(* IEC 61131-3 sources: SmartHomeNew/snapshots/2026-05-25 (part 3) *)

(* ---- FB_Heating_RootCause_Diagnostics.st ---- *)
// ==============================================================================
// Heating root-cause diagnostics observer
// Public diagnostics/explainability layer.
// Does NOT own control/runtime decisions.
// ==============================================================================
FUNCTION_BLOCK FB_Heating_RootCause_Diagnostics
VAR_INPUT
    VI_Enable : BOOL;
END_VAR
VAR
    fbRootCause : FB_Diagnostics_RootCause;
    fbDemandMap : FB_Heating_Demand_Map;
    L_Demand_Map : ARRAY[1..GVL_CONSTANTS.C_MAX_MANIFOLDS] OF BOOL;
END_VAR

IF NOT VI_Enable THEN
    GVL_STATE.G_Heating_RootCause := E_Heating_RootCause.RC_NONE;
    GVL_STATE.G_Heating_RootConfidence := 0.0;
    GVL_STATE.G_Heating_Confidence := 0.0;
    GVL_STATE.G_Heating_Error_Score := 1.0;
    GVL_STATE.G_Heating_Confidence_Reason_Code := -1;
    GVL_STATE.G_Heating_Confidence_Reason_Text := 'Heating diagnostics disabled';
    RETURN;
END_IF;

// ======================================================
// DEMAND MAP
// ======================================================
fbDemandMap(
    VI_Zone_Valves := GVL_STATE.G_Zone_Valves,
    VI_Zone_Configs := GVL_CONFIG.G_HMI_FloorHeating_Configs,
    VO_Manifold_Demand_Map => L_Demand_Map
);

// ======================================================
// INTERNAL INFERENCE ENGINE
// ======================================================
fbRootCause(
    VI_Emergency_Stop := GVL_STATE.G_Safety_Emergency_Stop,
    VI_Gas_Safety := GVL_STATE.G_Safety_Gas_Latched,
    VI_IO_Failsafe := GVL_STATE.G_Heating_IO_Fault,

    VI_Cascade_Available := GVL_STATE.G_Heating_Cascade_Available,
    VI_Cascade_Degraded := GVL_STATE.G_Heating_Cascade_Degraded,
    VI_Cascade_Partial_Capacity := GVL_STATE.G_Heating_Cascade_Partial_Capacity,
    VI_Cascade_No_Flame := GVL_STATE.G_Heating_Cascade_No_Flame,
    VI_Cascade_Transport_Degraded := GVL_STATE.G_Heating_Cascade_Transport_Degraded,
    VI_Cascade_Ignition_Timeout := GVL_STATE.G_Heating_Cascade_Ignition_Timeout,
    VI_Cascade_Active_Boilers := GVL_STATE.G_Heating_Cascade_Active_Boilers,
    VI_Cascade_Available_Boilers := GVL_STATE.G_Heating_Cascade_Available_Boilers,

    VI_Boiler_OT_Online := GVL_STATE.G_Boiler_OT_Online,
    VI_Boiler_Error := GVL_STATE.G_Boiler_Error,
    VI_Boiler_Flame := GVL_STATE.G_Boiler_Flame,
    VI_Boiler_OT_Command_Timeout := GVL_STATE.G_Boiler_OT_Command_Timeout,
    VI_Boiler_OT_Heartbeat_Timeout := GVL_STATE.G_Boiler_OT_Heartbeat_Timeout,
    VI_Boiler_OT_Adapter_Error := GVL_STATE.G_Boiler_OT_Adapter_Error,

    VI_Manifold_Pumps := GVL_STATE.G_Manifold_Pumps,
    VI_Manifold_Valves := GVL_STATE.G_Manifold_Valves,

    VI_Sensor_Error := GVL_STATE.G_Heating_Sensor_Fault,
    VI_Supply_Temps := GVL_STATE.G_Manifold_T_Supply,
    VI_Target_Supply := GVL_STATE.G_Target_Temperature,
    VI_Demand_Map := L_Demand_Map
);

// ======================================================
// PUBLIC DIAGNOSTICS STATE
// ======================================================
GVL_STATE.G_Heating_RootCause := fbRootCause.VO_RootCause;
GVL_STATE.G_Heating_RootConfidence := fbRootCause.VO_Confidence;
GVL_STATE.G_Heating_Confidence := fbRootCause.VO_Confidence;
GVL_STATE.G_Heating_Error_Score := fbRootCause.VO_Error_Score;
GVL_STATE.G_Heating_Confidence_Reason_Code := fbRootCause.VO_Reason_Code;
GVL_STATE.G_Heating_Confidence_Reason_Text := fbRootCause.VO_Reason_Text;

END_FUNCTION_BLOCK
// >>> BULK_SYNC_ANCHOR: FB_Heating_RootCause_Diagnostics <<<

(* ---- FB_Heating_Runtime_Event_Manager.st ---- *)
// ==============================================================================
// Heating runtime event manager
// Read-only orchestration telemetry/event layer.
// DOES NOT own runtime.
// DOES NOT own heating logic.
// DOES NOT own diagnostics.
// DOES NOT own OpenTherm transport.
// ==============================================================================
FUNCTION_BLOCK FB_Heating_Runtime_Event_Manager
VAR_INPUT
    VI_Enable : BOOL;
    VI_Event : ST_Heating_Runtime_Phase_Event;
END_VAR
VAR_IN_OUT
    VIO_Buffer : ST_Heating_Runtime_Event_Buffer;
END_VAR
VAR_OUTPUT
    VO_Event_Stored : BOOL;
    VO_Buffer_Overflow : BOOL;
    VO_Manager_Ready : BOOL;
    VO_Manager_Status_Code : UINT;
    VO_Manager_Status_Text : STRING(128);
END_VAR
VAR
    L_Write_Index : UINT;
END_VAR

// ======================================================
// DEFAULTS
// ======================================================
VO_Event_Stored := FALSE;
VO_Buffer_Overflow := FALSE;
VO_Manager_Ready := FALSE;
VO_Manager_Status_Code := 0;
VO_Manager_Status_Text := 'Heating runtime event manager disabled';

IF NOT VI_Enable THEN
    RETURN;
END_IF;

// ======================================================
// BUFFER VALIDATION
// ======================================================
IF VIO_Buffer.Write_Index > 32 THEN
    VIO_Buffer.Write_Index := 1;
END_IF;

IF VIO_Buffer.Read_Index > 32 THEN
    VIO_Buffer.Read_Index := 1;
END_IF;

// ======================================================
// WRITE INDEX
// ======================================================
L_Write_Index := VIO_Buffer.Write_Index + 1;

IF L_Write_Index > 32 THEN
    L_Write_Index := 1;
END_IF;

// ======================================================
// STORE EVENT
// ======================================================
VIO_Buffer.Events[L_Write_Index] := VI_Event;
VIO_Buffer.Write_Index := L_Write_Index;

IF VIO_Buffer.Event_Count < 32 THEN
    VIO_Buffer.Event_Count := VIO_Buffer.Event_Count + 1;
ELSE
    VIO_Buffer.Overflow := TRUE;
    VO_Buffer_Overflow := TRUE;
END_IF;

// ======================================================
// BUFFER INTEGRITY
// ======================================================
VIO_Buffer.Ordering_Integrity_Valid :=
    VI_Event.Ordering_Valid;

VIO_Buffer.Isolation_Integrity_Valid :=
    VI_Event.Isolation_Valid;

VIO_Buffer.Diagnostics_Visibility_Valid :=
    VI_Event.Diagnostics_Visible;

VIO_Buffer.Explainability_Visibility_Valid :=
    VI_Event.Explainability_Visible;

VIO_Buffer.OpenTherm_Ownership_Valid :=
    VI_Event.OpenTherm_Ownership_Valid;

VIO_Buffer.Cascade_Ownership_Valid :=
    VI_Event.Cascade_Ownership_Valid;

VIO_Buffer.Safety_Ownership_Valid :=
    VI_Event.Safety_Integrity_Valid;

VIO_Buffer.Lifecycle_Integrity_Valid :=
    NOT VI_Event.Event_Failed;

// ======================================================
// BUFFER STATUS
// ======================================================
IF VO_Buffer_Overflow THEN
    VIO_Buffer.Status_Code := 100;
    VIO_Buffer.Status_Text := 'Heating runtime event buffer overflow';
ELSE
    VIO_Buffer.Status_Code := 1;
    VIO_Buffer.Status_Text := 'Heating runtime event stored';
END_IF;

// ======================================================
// OUTPUT STATUS
// ======================================================
VO_Event_Stored := TRUE;
VO_Manager_Ready := TRUE;
VO_Manager_Status_Code := VIO_Buffer.Status_Code;
VO_Manager_Status_Text := VIO_Buffer.Status_Text;

END_FUNCTION_BLOCK
// >>> BULK_SYNC_ANCHOR: FB_Heating_Runtime_Event_Manager <<<

(* ---- FB_Heating_Runtime_Observer.st ---- *)
// ==============================================================================
// Heating runtime observer
// Minimal observer-only runtime attachment.
// Read-only.
// Governance-locked.
// Finalized-state observation only.
// ==============================================================================
FUNCTION_BLOCK FB_Heating_Runtime_Observer
VAR_INPUT
    VI_Enable : BOOL;
    VI_Runtime_Context : ST_Heating_Runtime_Context;
    VI_Diagnostics_Valid : BOOL;
END_VAR
VAR_OUTPUT
    VO_Observation : ST_Heating_Runtime_Observation;

    VO_Observer_Ready : BOOL;
    VO_Observer_Fault : BOOL;
    VO_Status_Code : UINT;
    VO_Status_Text : STRING(128);
END_VAR

// ======================================================
// DEFAULTS
// ======================================================
VO_Observation.Runtime_Active := FALSE;
VO_Observation.Runtime_Ready := FALSE;
VO_Observation.Runtime_Fault := FALSE;
VO_Observation.Current_Phase := E_Heating_Runtime_Phase.HRP_DISABLED;

VO_Observation.DHW_Demand_Active := FALSE;
VO_Observation.DHW_Heating_Active := FALSE;
VO_Observation.DHW_Circulation_Active := FALSE;

VO_Observation.Heating_Demand_Active := FALSE;
VO_Observation.Heating_Runtime_Active := FALSE;
VO_Observation.Heating_Output_Active := FALSE;

VO_Observation.Cascade_Available := FALSE;
VO_Observation.Cascade_Degraded := FALSE;
VO_Observation.Cascade_Active_Boilers := 0;
VO_Observation.Cascade_Available_Boilers := 0;

VO_Observation.OpenTherm_Online := FALSE;
VO_Observation.OpenTherm_Command_Valid := FALSE;
VO_Observation.OpenTherm_Transport_Degraded := FALSE;

VO_Observation.Diagnostics_Active := FALSE;
VO_Observation.Explainability_Active := FALSE;

VO_Observation.DHW_Before_Heating_Observed := FALSE;
VO_Observation.Diagnostics_After_Publication_Observed := FALSE;
VO_Observation.Output_Projection_Last_Observed := FALSE;

VO_Observation.Runtime_Ownership_Valid := TRUE;
VO_Observation.Diagnostics_Ownership_Valid := TRUE;
VO_Observation.OpenTherm_Ownership_Valid := TRUE;
VO_Observation.Cascade_Ownership_Valid := TRUE;
VO_Observation.Safety_Ownership_Valid := TRUE;

VO_Observation.Observation_Status_Code := 0;
VO_Observation.Observation_Status_Text := 'Heating runtime observer disabled';

VO_Observer_Ready := FALSE;
VO_Observer_Fault := FALSE;
VO_Status_Code := 0;
VO_Status_Text := 'Heating runtime observer disabled';

IF NOT VI_Enable THEN
    RETURN;
END_IF;

// ======================================================
// FINALIZED-STATE OBSERVATION ONLY
// ======================================================
VO_Observation.Runtime_Active := VI_Runtime_Context.Runtime_Enabled;
VO_Observation.Runtime_Ready := VI_Runtime_Context.Runtime_Ready;
VO_Observation.Runtime_Fault := VI_Runtime_Context.Runtime_Fault;
VO_Observation.Current_Phase := VI_Runtime_Context.Current_Phase;

VO_Observation.Diagnostics_Active := VI_Diagnostics_Valid;
VO_Observation.Explainability_Active := VI_Runtime_Context.Explainability_Isolation_Valid;

VO_Observation.DHW_Before_Heating_Observed :=
    VI_Runtime_Context.DHW_Before_Heating_Valid;

VO_Observation.Diagnostics_After_Publication_Observed :=
    VI_Runtime_Context.State_Publication_Before_Diagnostics_Valid;

VO_Observation.Output_Projection_Last_Observed :=
    VI_Runtime_Context.Output_Projection_Last_Valid;

VO_Observation.Runtime_Ownership_Valid := TRUE;
VO_Observation.Diagnostics_Ownership_Valid :=
    VI_Runtime_Context.Diagnostics_Isolation_Valid;

VO_Observation.OpenTherm_Ownership_Valid :=
    VI_Runtime_Context.OpenTherm_Ownership_Valid;

VO_Observation.Cascade_Ownership_Valid :=
    VI_Runtime_Context.Cascade_Ownership_Valid;

VO_Observation.Safety_Ownership_Valid :=
    VI_Runtime_Context.Safety_Isolation_Valid;

// These domain-specific runtime values remain intentionally FALSE/0 here.
// They must be populated only by finalized publication contracts, not by internal runtime scans.
VO_Observation.DHW_Demand_Active := FALSE;
VO_Observation.DHW_Heating_Active := FALSE;
VO_Observation.DHW_Circulation_Active := FALSE;
VO_Observation.Heating_Demand_Active := FALSE;
VO_Observation.Heating_Runtime_Active := FALSE;
VO_Observation.Heating_Output_Active := FALSE;
VO_Observation.Cascade_Available := FALSE;
VO_Observation.Cascade_Degraded := FALSE;
VO_Observation.Cascade_Active_Boilers := 0;
VO_Observation.Cascade_Available_Boilers := 0;
VO_Observation.OpenTherm_Online := FALSE;
VO_Observation.OpenTherm_Command_Valid := FALSE;
VO_Observation.OpenTherm_Transport_Degraded := FALSE;

// ======================================================
// STATUS
// ======================================================
IF VI_Runtime_Context.Runtime_Fault THEN
    VO_Observation.Observation_Status_Code := 900;
    VO_Observation.Observation_Status_Text := 'Heating runtime observer detected runtime fault';

ELSIF NOT VI_Diagnostics_Valid THEN
    VO_Observation.Observation_Status_Code := 200;
    VO_Observation.Observation_Status_Text := 'Heating runtime diagnostics publication invalid';

ELSE
    VO_Observation.Observation_Status_Code := 1;
    VO_Observation.Observation_Status_Text := 'Heating runtime observer nominal';
END_IF;

VO_Observer_Ready := TRUE;
VO_Observer_Fault := FALSE;

VO_Status_Code := VO_Observation.Observation_Status_Code;
VO_Status_Text := VO_Observation.Observation_Status_Text;

END_FUNCTION_BLOCK
// >>> BULK_SYNC_ANCHOR: FB_Heating_Runtime_Observer <<<

(* ---- FB_Heating_Runtime_Observer_Authorization.st ---- *)
// ==============================================================================
// Heating runtime observer authorization
// Governed passive-bootstrap authorization only.
// Read-only.
// Deterministic.
// ==============================================================================
FUNCTION_BLOCK FB_Heating_Runtime_Observer_Authorization
VAR_INPUT
    VI_Enable_Request : BOOL;

    VI_Bootstrap_Mode : BOOL;
    VI_Passive_Mode : BOOL;
    VI_ReadOnly_Mode : BOOL;

    VI_Governance_Locked : BOOL;
    VI_Runtime_Authority_Disabled : BOOL;
    VI_Writable_Exports_Disabled : BOOL;
END_VAR
VAR_OUTPUT
    VO_Enable_Authorized : BOOL;
    VO_Enable_Effective : BOOL;

    VO_Authorization_Valid : BOOL;

    VO_Status_Code : UINT;
    VO_Status_Text : STRING(128);
END_VAR

// ======================================================
// DEFAULTS
// ======================================================
VO_Enable_Authorized := FALSE;
VO_Enable_Effective := FALSE;
VO_Authorization_Valid := FALSE;

VO_Status_Code := 0;
VO_Status_Text := 'Heating runtime observer authorization inactive';

// ======================================================
// REQUEST VALIDATION
// ======================================================
IF NOT VI_Enable_Request THEN
    RETURN;
END_IF;

// ======================================================
// GOVERNANCE VALIDATION
// ======================================================
IF NOT VI_Bootstrap_Mode THEN
    VO_Status_Code := 100;
    VO_Status_Text := 'Bootstrap mode required for observer authorization';
    RETURN;
END_IF;

IF NOT VI_Passive_Mode THEN
    VO_Status_Code := 110;
    VO_Status_Text := 'Passive mode required for observer authorization';
    RETURN;
END_IF;

IF NOT VI_ReadOnly_Mode THEN
    VO_Status_Code := 120;
    VO_Status_Text := 'Read-only mode required for observer authorization';
    RETURN;
END_IF;

IF NOT VI_Governance_Locked THEN
    VO_Status_Code := 130;
    VO_Status_Text := 'Governance lock required for observer authorization';
    RETURN;
END_IF;

IF NOT VI_Runtime_Authority_Disabled THEN
    VO_Status_Code := 140;
    VO_Status_Text := 'Runtime authority isolation required';
    RETURN;
END_IF;

IF NOT VI_Writable_Exports_Disabled THEN
    VO_Status_Code := 150;
    VO_Status_Text := 'Writable exports must remain disabled';
    RETURN;
END_IF;

// ======================================================
// AUTHORIZED PASSIVE BOOTSTRAP ACTIVATION
// ======================================================
VO_Enable_Authorized := TRUE;
VO_Enable_Effective := TRUE;
VO_Authorization_Valid := TRUE;

VO_Status_Code := 1;
VO_Status_Text := 'Heating runtime observer authorization granted';

END_FUNCTION_BLOCK
// >>> BULK_SYNC_ANCHOR: FB_Heating_Runtime_Observer_Authorization <<<

(* ---- FB_Heating_Runtime_Observer_Phase.st ---- *)
// ==============================================================================
// Heating runtime observer phase
// Owns governed observer authorization and finalized-state observer publication.
// Does NOT own heating control or output decisions.
// ==============================================================================
FUNCTION_BLOCK FB_Heating_Runtime_Observer_Phase
VAR_INPUT
    VI_Authorization_Stage : BOOL;
    VI_Finalization_Stage : BOOL;
    VI_Runtime_Context : ST_Heating_Runtime_Context;
    VI_Diagnostics_Valid : BOOL;
END_VAR
VAR_OUTPUT
    VO_Authorization_Executed : BOOL;
    VO_Finalization_Executed : BOOL;
    VO_Observer_Valid : BOOL;
END_VAR
VAR
    fbRuntimeObserver : FB_Heating_Runtime_Observer;
    fbRuntimeObserverAuthorization : FB_Heating_Runtime_Observer_Authorization;
    L_Enable_Last : BOOL := FALSE;
    L_Activation_Stabilized : BOOL := FALSE;
END_VAR

VO_Authorization_Executed := FALSE;
VO_Finalization_Executed := FALSE;
VO_Observer_Valid := FALSE;

// ======================================================
// GOVERNED OBSERVER AUTHORIZATION EVALUATION
// ======================================================
IF VI_Authorization_Stage THEN

    GVL_Heating_Runtime_Observer.G_Runtime_Observer_Lifecycle_State :=
        E_Runtime_Observer_Lifecycle_State.ROS_AUTHORIZATION_PENDING;
    GVL_Heating_Runtime_Observation.G_Runtime_Observer_Lifecycle_State :=
        E_Runtime_Observer_Lifecycle_State.ROS_AUTHORIZATION_PENDING;
    GVL_Heating_Runtime_Observation.G_Runtime_Observer_Lifecycle_Code := 10;
    GVL_Heating_Runtime_Observation.G_Runtime_Observer_Lifecycle_Text :=
        'Heating runtime observer authorization pending';
    GVL_Heating_Runtime_Observation.G_Runtime_Observer_Commissioning_Active :=
        GVL_Heating_Runtime_Observer.G_Runtime_Observer_Enable_Request;

    fbRuntimeObserverAuthorization(
        VI_Enable_Request := GVL_Heating_Runtime_Observer.G_Runtime_Observer_Enable_Request,
        VI_Bootstrap_Mode := GVL_Heating_Runtime_Observer.G_Runtime_Observer_Bootstrap_Mode,
        VI_Passive_Mode := GVL_Heating_Runtime_Observer.G_Runtime_Observer_Passive_Mode,
        VI_ReadOnly_Mode := GVL_Heating_Runtime_Observer.G_Runtime_Observer_ReadOnly_Mode,
        VI_Governance_Locked := GVL_Heating_Runtime_Observer.G_Runtime_Observer_Governance_Locked,
        VI_Runtime_Authority_Disabled := GVL_Heating_Runtime_Observer.G_Runtime_Observer_Runtime_Authority_Disabled,
        VI_Writable_Exports_Disabled := GVL_Heating_Runtime_Observer.G_Runtime_Observer_Writable_Exports_Disabled
    );

    GVL_Heating_Runtime_Observer.G_Runtime_Observer_Enable_Authorized :=
        fbRuntimeObserverAuthorization.VO_Enable_Authorized;

    GVL_Heating_Runtime_Observer.G_Runtime_Observer_Enable_Effective :=
        fbRuntimeObserverAuthorization.VO_Enable_Effective;

    GVL_Heating_Runtime_Observer.G_Runtime_Observer_Authorization_Valid :=
        fbRuntimeObserverAuthorization.VO_Authorization_Valid;

    GVL_Heating_Runtime_Observer.G_Runtime_Observer_Authorization_Status_Code :=
        fbRuntimeObserverAuthorization.VO_Status_Code;

    GVL_Heating_Runtime_Observer.G_Runtime_Observer_Authorization_Status_Text :=
        fbRuntimeObserverAuthorization.VO_Status_Text;

    IF NOT GVL_Heating_Runtime_Observer.G_Runtime_Observer_Enable_Request THEN
        GVL_Heating_Runtime_Observer.G_Runtime_Observer_Lifecycle_State :=
            E_Runtime_Observer_Lifecycle_State.ROS_INACTIVE;
        GVL_Heating_Runtime_Observation.G_Runtime_Observer_Lifecycle_State :=
            E_Runtime_Observer_Lifecycle_State.ROS_INACTIVE;
        GVL_Heating_Runtime_Observation.G_Runtime_Observer_Lifecycle_Code := 0;
        GVL_Heating_Runtime_Observation.G_Runtime_Observer_Lifecycle_Text :=
            'Heating runtime observer inactive';
        GVL_Heating_Runtime_Observation.G_Runtime_Observer_Commissioning_Active := FALSE;
    ELSIF NOT GVL_Heating_Runtime_Observer.G_Runtime_Observer_Enable_Effective THEN
        GVL_Heating_Runtime_Observer.G_Runtime_Observer_Lifecycle_State :=
            E_Runtime_Observer_Lifecycle_State.ROS_AUTHORIZATION_DENIED;
        GVL_Heating_Runtime_Observation.G_Runtime_Observer_Lifecycle_State :=
            E_Runtime_Observer_Lifecycle_State.ROS_AUTHORIZATION_DENIED;
        GVL_Heating_Runtime_Observation.G_Runtime_Observer_Lifecycle_Code := 20;
        GVL_Heating_Runtime_Observation.G_Runtime_Observer_Lifecycle_Text :=
            'Heating runtime observer authorization denied';
    END_IF;

    VO_Authorization_Executed := TRUE;
END_IF;

// ======================================================
// GOVERNED FINALIZED-STATE RUNTIME OBSERVER
// ======================================================
IF VI_Finalization_Stage THEN

    IF GVL_Heating_Runtime_Observer.G_Runtime_Observer_Enable_Effective THEN

        GVL_Heating_Runtime_Observer.G_Runtime_Observer_Rollback_Validated := FALSE;

        IF NOT L_Enable_Last THEN
            L_Activation_Stabilized := FALSE;

            GVL_Heating_Runtime_Observer.G_Runtime_Observer_Lifecycle_State :=
                E_Runtime_Observer_Lifecycle_State.ROS_STABILIZATION;
            GVL_Heating_Runtime_Observation.G_Runtime_Observer_Lifecycle_State :=
                E_Runtime_Observer_Lifecycle_State.ROS_STABILIZATION;
            GVL_Heating_Runtime_Observation.G_Runtime_Observer_Lifecycle_Code := 30;
            GVL_Heating_Runtime_Observation.G_Runtime_Observer_Lifecycle_Text :=
                'Heating runtime observer stabilization active';

            GVL_Heating_Runtime_Observation.G_Runtime_Observer_Commissioning_Required := TRUE;
            GVL_Heating_Runtime_Observation.G_Runtime_Observer_Commissioning_Active := TRUE;
            GVL_Heating_Runtime_Observation.G_Runtime_Observer_Commissioning_Complete := FALSE;

            GVL_Heating_Runtime_Observation.G_Runtime_Observation_Publication_Valid := FALSE;
            GVL_Heating_Runtime_Observation.G_Runtime_Observation_Stabilization_Complete := FALSE;
            GVL_Heating_Runtime_Observation.G_Runtime_Observation_Operational := FALSE;

            GVL_Heating_Runtime_Observation.G_Runtime_Observation_Valid := FALSE;
            GVL_Heating_Runtime_Observation.G_Runtime_Observer_Ready := FALSE;
            GVL_Heating_Runtime_Observation.G_Runtime_Observer_Fault := FALSE;
            GVL_Heating_Runtime_Observation.G_Runtime_Observation_Status_Code := 100;
            GVL_Heating_Runtime_Observation.G_Runtime_Observation_Status_Text :=
                'Heating runtime observer stabilization cycle active';
        END_IF;

        fbRuntimeObserver(
            VI_Enable := TRUE,
            VI_Runtime_Context := VI_Runtime_Context,
            VI_Diagnostics_Valid := VI_Diagnostics_Valid
        );

        GVL_Heating_Runtime_Observation.G_Runtime_Observation :=
            fbRuntimeObserver.VO_Observation;

        IF L_Activation_Stabilized THEN
            GVL_Heating_Runtime_Observer.G_Runtime_Observer_Lifecycle_State :=
                E_Runtime_Observer_Lifecycle_State.ROS_OPERATIONAL;
            GVL_Heating_Runtime_Observation.G_Runtime_Observer_Lifecycle_State :=
                E_Runtime_Observer_Lifecycle_State.ROS_OPERATIONAL;
            GVL_Heating_Runtime_Observation.G_Runtime_Observer_Lifecycle_Code := 40;
            GVL_Heating_Runtime_Observation.G_Runtime_Observer_Lifecycle_Text :=
                'Heating runtime observer operational';

            GVL_Heating_Runtime_Observation.G_Runtime_Observer_Commissioning_Required := FALSE;
            GVL_Heating_Runtime_Observation.G_Runtime_Observer_Commissioning_Active := FALSE;
            GVL_Heating_Runtime_Observation.G_Runtime_Observer_Commissioning_Complete := TRUE;

            GVL_Heating_Runtime_Observation.G_Runtime_Observation_Publication_Valid := TRUE;
            GVL_Heating_Runtime_Observation.G_Runtime_Observation_Stabilization_Complete := TRUE;
            GVL_Heating_Runtime_Observation.G_Runtime_Observation_Operational := TRUE;

            GVL_Heating_Runtime_Observation.G_Runtime_Observation_Valid := TRUE;
            GVL_Heating_Runtime_Observation.G_Runtime_Observer_Ready :=
                fbRuntimeObserver.VO_Observer_Ready;
            GVL_Heating_Runtime_Observation.G_Runtime_Observer_Fault :=
                fbRuntimeObserver.VO_Observer_Fault;
            GVL_Heating_Runtime_Observation.G_Runtime_Observation_Status_Code :=
                fbRuntimeObserver.VO_Status_Code;
            GVL_Heating_Runtime_Observation.G_Runtime_Observation_Status_Text :=
                fbRuntimeObserver.VO_Status_Text;

            GVL_Heating_Runtime_Observer.G_Runtime_Observer_Activation_Validated := TRUE;
            GVL_Heating_Runtime_Observer.G_Runtime_Observer_Sequencing_Validated := TRUE;
            GVL_Heating_Runtime_Observer.G_Runtime_Observer_Publication_Validated := TRUE;
            VO_Observer_Valid := TRUE;
        ELSE
            L_Activation_Stabilized := TRUE;
        END_IF;

    ELSE
        L_Activation_Stabilized := FALSE;

        IF L_Enable_Last THEN
            GVL_Heating_Runtime_Observer.G_Runtime_Observer_Lifecycle_State :=
                E_Runtime_Observer_Lifecycle_State.ROS_ROLLBACK;
            GVL_Heating_Runtime_Observation.G_Runtime_Observer_Lifecycle_State :=
                E_Runtime_Observer_Lifecycle_State.ROS_ROLLBACK;
            GVL_Heating_Runtime_Observation.G_Runtime_Observer_Lifecycle_Code := 50;
            GVL_Heating_Runtime_Observation.G_Runtime_Observer_Lifecycle_Text :=
                'Heating runtime observer rollback cleanup completed';
        ELSIF GVL_Heating_Runtime_Observer.G_Runtime_Observer_Enable_Request THEN
            GVL_Heating_Runtime_Observer.G_Runtime_Observer_Lifecycle_State :=
                E_Runtime_Observer_Lifecycle_State.ROS_AUTHORIZATION_DENIED;
            GVL_Heating_Runtime_Observation.G_Runtime_Observer_Lifecycle_State :=
                E_Runtime_Observer_Lifecycle_State.ROS_AUTHORIZATION_DENIED;
            GVL_Heating_Runtime_Observation.G_Runtime_Observer_Lifecycle_Code := 20;
            GVL_Heating_Runtime_Observation.G_Runtime_Observer_Lifecycle_Text :=
                'Heating runtime observer authorization denied';
        ELSE
            GVL_Heating_Runtime_Observer.G_Runtime_Observer_Lifecycle_State :=
                E_Runtime_Observer_Lifecycle_State.ROS_INACTIVE;
            GVL_Heating_Runtime_Observation.G_Runtime_Observer_Lifecycle_State :=
                E_Runtime_Observer_Lifecycle_State.ROS_INACTIVE;
            GVL_Heating_Runtime_Observation.G_Runtime_Observer_Lifecycle_Code := 0;
            GVL_Heating_Runtime_Observation.G_Runtime_Observer_Lifecycle_Text :=
                'Heating runtime observer inactive';
        END_IF;

        GVL_Heating_Runtime_Observation.G_Runtime_Observer_Commissioning_Required := TRUE;
        GVL_Heating_Runtime_Observation.G_Runtime_Observer_Commissioning_Active := FALSE;
        GVL_Heating_Runtime_Observation.G_Runtime_Observer_Commissioning_Complete := FALSE;

        GVL_Heating_Runtime_Observation.G_Runtime_Observation.Runtime_Active := FALSE;
        GVL_Heating_Runtime_Observation.G_Runtime_Observation.Runtime_Ready := FALSE;
        GVL_Heating_Runtime_Observation.G_Runtime_Observation.Runtime_Fault := FALSE;
        GVL_Heating_Runtime_Observation.G_Runtime_Observation.Current_Phase := E_Heating_Runtime_Phase.HRP_DISABLED;

        GVL_Heating_Runtime_Observation.G_Runtime_Observation.DHW_Demand_Active := FALSE;
        GVL_Heating_Runtime_Observation.G_Runtime_Observation.DHW_Heating_Active := FALSE;
        GVL_Heating_Runtime_Observation.G_Runtime_Observation.DHW_Circulation_Active := FALSE;

        GVL_Heating_Runtime_Observation.G_Runtime_Observation.Heating_Demand_Active := FALSE;
        GVL_Heating_Runtime_Observation.G_Runtime_Observation.Heating_Runtime_Active := FALSE;
        GVL_Heating_Runtime_Observation.G_Runtime_Observation.Heating_Output_Active := FALSE;

        GVL_Heating_Runtime_Observation.G_Runtime_Observation.Cascade_Available := FALSE;
        GVL_Heating_Runtime_Observation.G_Runtime_Observation.Cascade_Degraded := FALSE;
        GVL_Heating_Runtime_Observation.G_Runtime_Observation.Cascade_Active_Boilers := 0;
        GVL_Heating_Runtime_Observation.G_Runtime_Observation.Cascade_Available_Boilers := 0;

        GVL_Heating_Runtime_Observation.G_Runtime_Observation.OpenTherm_Online := FALSE;
        GVL_Heating_Runtime_Observation.G_Runtime_Observation.OpenTherm_Command_Valid := FALSE;
        GVL_Heating_Runtime_Observation.G_Runtime_Observation.OpenTherm_Transport_Degraded := FALSE;

        GVL_Heating_Runtime_Observation.G_Runtime_Observation.Diagnostics_Active := FALSE;
        GVL_Heating_Runtime_Observation.G_Runtime_Observation.Explainability_Active := FALSE;

        GVL_Heating_Runtime_Observation.G_Runtime_Observation.DHW_Before_Heating_Observed := FALSE;
        GVL_Heating_Runtime_Observation.G_Runtime_Observation.Diagnostics_After_Publication_Observed := FALSE;
        GVL_Heating_Runtime_Observation.G_Runtime_Observation.Output_Projection_Last_Observed := FALSE;

        GVL_Heating_Runtime_Observation.G_Runtime_Observation.Runtime_Ownership_Valid := FALSE;
        GVL_Heating_Runtime_Observation.G_Runtime_Observation.Diagnostics_Ownership_Valid := FALSE;
        GVL_Heating_Runtime_Observation.G_Runtime_Observation.OpenTherm_Ownership_Valid := FALSE;
        GVL_Heating_Runtime_Observation.G_Runtime_Observation.Cascade_Ownership_Valid := FALSE;
        GVL_Heating_Runtime_Observation.G_Runtime_Observation.Safety_Ownership_Valid := FALSE;

        GVL_Heating_Runtime_Observation.G_Runtime_Observation.Observation_Status_Code := 0;
        GVL_Heating_Runtime_Observation.G_Runtime_Observation.Observation_Status_Text :=
            'Heating runtime observation inactive';

        GVL_Heating_Runtime_Observation.G_Runtime_Observation_Publication_Valid := FALSE;
        GVL_Heating_Runtime_Observation.G_Runtime_Observation_Stabilization_Complete := FALSE;
        GVL_Heating_Runtime_Observation.G_Runtime_Observation_Operational := FALSE;

        GVL_Heating_Runtime_Observation.G_Runtime_Observation_Valid := FALSE;
        GVL_Heating_Runtime_Observation.G_Runtime_Observer_Ready := FALSE;
        GVL_Heating_Runtime_Observation.G_Runtime_Observer_Fault := FALSE;
        GVL_Heating_Runtime_Observation.G_Runtime_Observation_Status_Code := 0;
        GVL_Heating_Runtime_Observation.G_Runtime_Observation_Status_Text :=
            'Heating runtime observation inactive';

        GVL_Heating_Runtime_Observer.G_Runtime_Observer_Activation_Validated := FALSE;
        GVL_Heating_Runtime_Observer.G_Runtime_Observer_Sequencing_Validated := FALSE;
        GVL_Heating_Runtime_Observer.G_Runtime_Observer_Publication_Validated := FALSE;
        GVL_Heating_Runtime_Observer.G_Runtime_Observer_Rollback_Validated := TRUE;
    END_IF;

    L_Enable_Last :=
        GVL_Heating_Runtime_Observer.G_Runtime_Observer_Enable_Effective;

    VO_Finalization_Executed := TRUE;
END_IF;

END_FUNCTION_BLOCK
// >>> BULK_SYNC_ANCHOR: FB_Heating_Runtime_Observer_Phase <<<

(* ---- FB_Heating_Runtime_OT_Cascade_Correlator.st ---- *)
// ==============================================================================
// Heating runtime OT and cascade correlator
// Read-only degradation correlation layer.
// ==============================================================================
FUNCTION_BLOCK FB_Heating_Runtime_OT_Cascade_Correlator
VAR_INPUT
    VI_Enable : BOOL;
    VI_Cascade_Degraded : BOOL;
    VI_OT_Degraded : BOOL;
    VI_OT_Command_Valid : BOOL;
    VI_Boiler_Count : UINT;
END_VAR
VAR_OUTPUT
    VO_Correlation_Detected : BOOL;
    VO_Status_Code : UINT;
    VO_Status_Text : STRING(128);
END_VAR

VO_Correlation_Detected := FALSE;
VO_Status_Code := 0;
VO_Status_Text := 'Heating OT/cascade correlator disabled';

IF NOT VI_Enable THEN
    RETURN;
END_IF;

VO_Correlation_Detected :=
    VI_Cascade_Degraded OR
    VI_OT_Degraded OR
    NOT VI_OT_Command_Valid OR
    (VI_Boiler_Count = 0);

IF VO_Correlation_Detected THEN
    VO_Status_Code := 200;
    VO_Status_Text := 'Heating OT/cascade degradation correlated';
ELSE
    VO_Status_Code := 1;
    VO_Status_Text := 'Heating OT/cascade nominal';
END_IF;

END_FUNCTION_BLOCK
// >>> BULK_SYNC_ANCHOR: FB_Heating_Runtime_OT_Cascade_Correlator <<<

(* ---- FB_Heating_Runtime_Supervisory_Publication_Adapter.st ---- *)
FUNCTION_BLOCK FB_Heating_Runtime_Supervisory_Publication_Adapter
VAR_INPUT
    VI_Enable : BOOL;
    VI_Predictive_State : ST_Heating_Runtime_Predictive_State;
    VI_Causality_Node : ST_Heating_Runtime_Causality_Node;
    VI_Causality_Edge : ST_Heating_Runtime_Causality_Edge;
    VI_Blackbox_Event : ST_Heating_Runtime_Blackbox_Event;
    VI_Anomaly : ST_Heating_Runtime_Anomaly;
END_VAR

IF NOT VI_Enable THEN
    RETURN;
END_IF;

GVL_Heating_Runtime_Supervisory_Publication.G_Publication.Supervisory_Visible := TRUE;
GVL_Heating_Runtime_Supervisory_Publication.G_Publication.Predictive_State := VI_Predictive_State;
GVL_Heating_Runtime_Supervisory_Publication.G_Publication.Source_Instability_Attention := VI_Predictive_State.Source_Instability_Attention;
GVL_Heating_Runtime_Supervisory_Publication.G_Publication.Source_Oscillation_Trend_Visible := VI_Predictive_State.Source_Oscillation_Trend_Visible;
GVL_Heating_Runtime_Supervisory_Publication.G_Publication.Runtime_Degraded := VI_Anomaly.Runtime_Degraded;
GVL_Heating_Runtime_Supervisory_Publication.G_Publication.Runtime_Fault := VI_Anomaly.Critical_Anomaly;
GVL_Heating_Runtime_Supervisory_Publication.G_Publication.Explainability_Degraded := VI_Anomaly.Explainability_Degraded;
GVL_Heating_Runtime_Supervisory_Publication.G_Publication.Diagnostics_Degraded := VI_Anomaly.Diagnostics_Degraded;
GVL_Heating_Runtime_Supervisory_Publication.G_Publication.Causality_Active := VI_Causality_Node.Node_Active;
GVL_Heating_Runtime_Supervisory_Publication.G_Publication.Propagation_Detected := VI_Causality_Edge.Propagation_Detected;
GVL_Heating_Runtime_Supervisory_Publication.G_Publication.Reconstruction_Visible := VI_Blackbox_Event.Event_Active;
GVL_Heating_Runtime_Supervisory_Publication.G_Publication.Status_Code := VI_Predictive_State.Status_Code;
GVL_Heating_Runtime_Supervisory_Publication.G_Publication.Status_Text := VI_Predictive_State.Status_Text;

END_FUNCTION_BLOCK

(* ---- FB_Heating_Safe_State.st ---- *)
FUNCTION_BLOCK FB_Heating_Safe_State
VAR_INPUT
    VI_Block_Normal_Heating : BOOL;
    VI_IO_Failsafe_Active : BOOL;
    VI_Gas_Safety_Active : BOOL;
    VI_Freeze_Active : BOOL;
    VI_Freeze_Target_Supply : REAL;
    VI_Manifold_Temps_Supply : ARRAY[1..GVL_CONSTANTS.C_MAX_MANIFOLDS] OF REAL;
    VI_Boiler_Error_Status : ARRAY[1..GVL_CONSTANTS.C_MAX_BOILERS] OF BOOL;
    VI_Boiler_OT_Online : ARRAY[1..GVL_CONSTANTS.C_MAX_BOILERS] OF BOOL;
END_VAR
VAR_OUTPUT
    VO_Applied : BOOL;
    VO_Zone_Valves : ARRAY[1..GVL_CONSTANTS.C_MAX_HEATING_CIRCUITS] OF BOOL;
    VO_Manifold_Pumps : ARRAY[1..GVL_CONSTANTS.C_MAX_MANIFOLDS] OF BOOL;
    VO_Manifold_Valves : ARRAY[1..GVL_CONSTANTS.C_MAX_MANIFOLDS] OF REAL;
    VO_Boiler_OT_Enable : ARRAY[1..GVL_CONSTANTS.C_MAX_BOILERS] OF BOOL;
    VO_Boiler_OT_Setpoint : ARRAY[1..GVL_CONSTANTS.C_MAX_BOILERS] OF REAL;
    VO_Boiler_Status : ARRAY[1..GVL_CONSTANTS.C_MAX_BOILERS] OF ST_Boiler_Status;
    VO_Backup_Circulation_Pump : BOOL;
    VO_Electric_Heater_Enable : BOOL;
    VO_Freeze_Risk_Status : BOOL;
END_VAR
VAR
    L_i : INT;
    L_Min_Supply_Temp : REAL;
    L_Freeze_Circulation_Required : BOOL;
    L_Empty_Boiler_Status : ST_Boiler_Status;
END_VAR

// Reset all retained FB outputs on every call.
// Safe-state FB instances keep VAR_OUTPUT values between scans unless overwritten.
VO_Applied := FALSE;
VO_Backup_Circulation_Pump := FALSE;
VO_Electric_Heater_Enable := FALSE;
VO_Freeze_Risk_Status := FALSE;

FOR L_i := 1 TO GVL_CONSTANTS.C_MAX_HEATING_CIRCUITS DO
    VO_Zone_Valves[L_i] := FALSE;
END_FOR;

FOR L_i := 1 TO GVL_CONSTANTS.C_MAX_MANIFOLDS DO
    VO_Manifold_Pumps[L_i] := FALSE;
    VO_Manifold_Valves[L_i] := REAL#0.0;
END_FOR;

FOR L_i := 1 TO GVL_CONSTANTS.C_MAX_BOILERS DO
    VO_Boiler_OT_Enable[L_i] := FALSE;
    VO_Boiler_OT_Setpoint[L_i] := REAL#0.0;
    VO_Boiler_Status[L_i] := L_Empty_Boiler_Status;
END_FOR;

VO_Applied := VI_Block_Normal_Heating;

L_Freeze_Circulation_Required := VI_Freeze_Active AND (VI_IO_Failsafe_Active OR VI_Gas_Safety_Active);

IF NOT VI_Block_Normal_Heating THEN
    RETURN;
END_IF;

// =============================
// ZONE VALVES (FIXED)
// =============================
FOR L_i := 1 TO GVL_CONSTANTS.C_MAX_HEATING_CIRCUITS DO
    IF L_Freeze_Circulation_Required THEN
        VO_Zone_Valves[L_i] := TRUE;
    ELSE
        VO_Zone_Valves[L_i] := FALSE;
    END_IF;
END_FOR;

// =============================
// MANIFOLD CONTROL
// =============================
FOR L_i := 1 TO GVL_CONSTANTS.C_MAX_MANIFOLDS DO
    IF L_Freeze_Circulation_Required THEN
        VO_Manifold_Pumps[L_i] := TRUE;
        VO_Manifold_Valves[L_i] := REAL#35.0;
    ELSE
        VO_Manifold_Pumps[L_i] := FALSE;
        VO_Manifold_Valves[L_i] := REAL#0.0;
    END_IF;
END_FOR;

// =============================
// BOILERS OFF
// =============================
FOR L_i := 1 TO GVL_CONSTANTS.C_MAX_BOILERS DO
    VO_Boiler_OT_Enable[L_i] := FALSE;
    VO_Boiler_OT_Setpoint[L_i] := REAL#0.0;
    VO_Boiler_Status[L_i].Warning := FALSE;
    VO_Boiler_Status[L_i].Error := TRUE;
END_FOR;

// =============================
// FREEZE PROTECTION LOGIC
// =============================
IF VI_Gas_Safety_Active AND VI_Freeze_Active THEN
    VO_Backup_Circulation_Pump := TRUE;

    L_Min_Supply_Temp := REAL#1000.0;
    FOR L_i := 1 TO GVL_CONSTANTS.C_MAX_MANIFOLDS DO
        IF VI_Manifold_Temps_Supply[L_i] < L_Min_Supply_Temp THEN
            L_Min_Supply_Temp := VI_Manifold_Temps_Supply[L_i];
        END_IF;
    END_FOR;

    IF L_Min_Supply_Temp > REAL#900.0 THEN
        L_Min_Supply_Temp := REAL#0.0;
    END_IF;

    IF L_Min_Supply_Temp < (VI_Freeze_Target_Supply - REAL#1.0) THEN
        VO_Electric_Heater_Enable := TRUE;
    ELSIF L_Min_Supply_Temp > (VI_Freeze_Target_Supply + REAL#1.0) THEN
        VO_Electric_Heater_Enable := FALSE;
    END_IF;

    VO_Freeze_Risk_Status := TRUE;
END_IF;

// =============================
// IO FAILSAFE + FREEZE
// =============================
IF VI_IO_Failsafe_Active AND VI_Freeze_Active THEN
    IF VI_Boiler_OT_Online[1] AND NOT VI_Boiler_Error_Status[1] THEN
        VO_Boiler_OT_Enable[1] := TRUE;
        VO_Boiler_OT_Setpoint[1] := VI_Freeze_Target_Supply;
    END_IF;
END_IF;

END_FUNCTION_BLOCK
// >>> BULK_SYNC_ANCHOR: FB_Heating_Safe_State <<<

(* ---- FB_Input_Quality_Observer.st ---- *)
FUNCTION_BLOCK FB_Input_Quality_Observer
VAR_INPUT
    VI_Enable : BOOL;
    VI_Value : REAL;
    VI_System_Time_MS : UDINT;
    VI_Spike_Threshold : REAL;
    VI_Stuck_Timeout_MS : UDINT;
END_VAR
VAR_OUTPUT
    VO_Quality : ST_Input_Quality_Record;
END_VAR
VAR
    L_Last_Value : REAL;
    L_Last_Change_MS : UDINT;
    L_Delta : REAL;
END_VAR

VO_Quality.Quality_Visible := VI_Enable;

IF NOT VI_Enable THEN
    RETURN;
END_IF;

VO_Quality.Value_Valid := TRUE;
VO_Quality.Value_Degraded := FALSE;
VO_Quality.Spike_Detected := FALSE;
VO_Quality.Stuck_Detected := FALSE;
VO_Quality.Confidence := REAL#1.0;
VO_Quality.Reason_Code := 0;
VO_Quality.Reason_Text := 'OK';

L_Delta := ABS(VI_Value - L_Last_Value);

IF L_Delta > VI_Spike_Threshold THEN
    VO_Quality.Spike_Detected := TRUE;
    VO_Quality.Value_Degraded := TRUE;
    VO_Quality.Confidence := REAL#0.4;
    VO_Quality.Reason_Code := 1;
    VO_Quality.Reason_Text := 'Spike detected';
END_IF;

IF L_Delta > REAL#0.05 THEN
    L_Last_Change_MS := VI_System_Time_MS;
END_IF;

IF (VI_System_Time_MS > L_Last_Change_MS) AND
   ((VI_System_Time_MS - L_Last_Change_MS) > VI_Stuck_Timeout_MS) THEN

    VO_Quality.Stuck_Detected := TRUE;
    VO_Quality.Value_Degraded := TRUE;

    IF VO_Quality.Confidence > REAL#0.6 THEN
        VO_Quality.Confidence := REAL#0.6;
    END_IF;

    IF VO_Quality.Reason_Code = 0 THEN
        VO_Quality.Reason_Code := 2;
        VO_Quality.Reason_Text := 'Sensor appears stuck';
    END_IF;
END_IF;

VO_Quality.Last_Value := VI_Value;
VO_Quality.Last_Change_MS := L_Last_Change_MS;

L_Last_Value := VI_Value;

END_FUNCTION_BLOCK

(* ---- FB_Modbus_Response_Apply.st ---- *)
FUNCTION_BLOCK FB_Modbus_Response_Apply
VAR_INPUT
    VI_Request_Valid : BOOL;
    VI_Request_Index : INT;
    VI_Request_Sequence : UDINT;
    VI_Parser_Valid : BOOL;
    VI_Parser_Error : BOOL;
    VI_Parser_Error_Code : WORD;
    VI_Register_Count : UINT;
    VI_Register_Value : ARRAY[1..32] OF WORD;
    VI_System_Time_MS : UDINT;
END_VAR

VAR_OUTPUT
    VO_Response_Applied : BOOL;
END_VAR

VAR
    L_i : INT;
    L_Count : INT;
END_VAR

// ======================================================
// MODBUS RESPONSE APPLY LAYER
// ======================================================
// Transfers validated parser result into bridge/master response.
//
// Safety principles:
//   - Only validated parser result may produce Done.
//   - Parser error produces Error response.
//   - No synthetic successful response.
// ======================================================

VO_Response_Applied := FALSE;

IF NOT VI_Request_Valid THEN
    RETURN;
END_IF;

IF (VI_Request_Index < 1) OR (VI_Request_Index > 16) THEN
    RETURN;
END_IF;

// ======================================================
// PARSER ERROR
// ======================================================
IF VI_Parser_Error THEN

    GVL_MODBUS_RTU_BRIDGE.G_Response_Busy := FALSE;
    GVL_MODBUS_RTU_BRIDGE.G_Response_Done := FALSE;
    GVL_MODBUS_RTU_BRIDGE.G_Response_Error := TRUE;
    GVL_MODBUS_RTU_BRIDGE.G_Response_Error_Code := VI_Parser_Error_Code;
    GVL_MODBUS_RTU_BRIDGE.G_Response_Sequence := VI_Request_Sequence;
    GVL_MODBUS_RTU_BRIDGE.G_Response_Update_MS := VI_System_Time_MS;

    VO_Response_Applied := TRUE;

    RETURN;
END_IF;

// ======================================================
// VALID PARSED RESPONSE
// ======================================================
IF VI_Parser_Valid THEN

    FOR L_i := 1 TO 32 DO
        GVL_MODBUS_RTU_BRIDGE.G_Response_Value[L_i] := 0;
    END_FOR;

    L_Count := UINT_TO_INT(VI_Register_Count);

    IF L_Count > 32 THEN
        L_Count := 32;
    END_IF;

    FOR L_i := 1 TO L_Count DO
        GVL_MODBUS_RTU_BRIDGE.G_Response_Value[L_i] :=
            VI_Register_Value[L_i];
    END_FOR;

    GVL_MODBUS_RTU_BRIDGE.G_Response_Busy := FALSE;
    GVL_MODBUS_RTU_BRIDGE.G_Response_Done := TRUE;
    GVL_MODBUS_RTU_BRIDGE.G_Response_Error := FALSE;
    GVL_MODBUS_RTU_BRIDGE.G_Response_Error_Code := 0;
    GVL_MODBUS_RTU_BRIDGE.G_Response_Sequence := VI_Request_Sequence;
    GVL_MODBUS_RTU_BRIDGE.G_Response_Update_MS := VI_System_Time_MS;

    VO_Response_Applied := TRUE;

END_IF;

END_FUNCTION_BLOCK

(* ---- FB_NVRAM_Manager.st ---- *)
FUNCTION_BLOCK FB_NVRAM_Manager
VAR_INPUT
    VI_Command                  : BYTE; // 1=WRITE (READ not implemented)
    VI_Offset                   : UDINT; // Смещение в байтах
    VI_DataRef                  : REFERENCE TO BYTE;
    VI_DataSize                 : UDINT; // КРИТИЧНО: используем этот размер вместо SIZEOF
    VI_System_Time_MS           : UDINT;
    VI_Operator_ID              : STRING(10);
    VI_IsActivePLC              : BOOL;
    VI_TwoPersonConfirmation    : BOOL;
END_VAR
VAR_OUTPUT
    VO_Done                     : BOOL;
    VO_Error                    : BOOL;
    VO_ErrorID                  : UDINT;
    // VO_ReadDataRef removed (REFERENCE TO not allowed in output)
    VO_HMI_Status_Message       : STRING(200);
END_VAR
VAR
    L_prev_Command              : BYTE;
    L_cmd_rising                : BOOL;
    L_i                         : UDINT;
    L_Data_Changed              : BOOL; // Флаг изменения данных
    L_pData                     : POINTER TO BYTE;
END_VAR
VAR CONSTANT
    // Must match GVL_Retain.G_NVRAM_Data upper bound + 1.
    // Active persistent snapshot currently writes 5 bytes; 512 bytes are kept
    // as conservative compact reserve for future settings records.
    C_MAX_NVRAM_SIZE            : UDINT := 512;
END_VAR

// Детекция фронта команды
L_cmd_rising := (VI_Command <> 0) AND (L_prev_Command = 0);
L_prev_Command := VI_Command;

IF L_cmd_rising THEN
    VO_Done := FALSE;
    VO_Error := FALSE;
    VO_ErrorID := 0;
    VO_HMI_Status_Message := '';

    // Валидация смещения
    IF VI_Offset >= C_MAX_NVRAM_SIZE THEN
        VO_Error := TRUE;
        VO_ErrorID := 16#1501;
        VO_HMI_Status_Message := 'NVRAM: Неверное смещение';
        VO_Done := TRUE;
        RETURN;
    END_IF;

    // Валидация указателя
    IF NOT __ISVALIDREF(VI_DataRef) THEN
        VO_Error := TRUE;
        VO_ErrorID := 16#150A;
        VO_HMI_Status_Message := 'NVRAM: Недействительная ссылка на данные';
        VO_Done := TRUE;
        RETURN;
    END_IF;

    L_pData := ADR(VI_DataRef);

    IF (VI_Offset + VI_DataSize) > C_MAX_NVRAM_SIZE THEN
        VO_Error := TRUE;
        VO_ErrorID := 16#150B;
        VO_HMI_Status_Message := 'NVRAM: Размер данных превышает доступный объем';
        VO_Done := TRUE;
        RETURN;
    END_IF;

    IF VI_Command = 2 THEN
        VO_Error := TRUE;
        VO_ErrorID := 16#150D;
        VO_HMI_Status_Message := 'NVRAM: READ not implemented';
        VO_Done := TRUE;
        RETURN;
    END_IF;

    IF VI_Command = 1 THEN // ЗАПИСЬ (WRITE)
        IF NOT VI_IsActivePLC THEN
            VO_Error := TRUE;
            VO_ErrorID := 16#1509;
            VO_HMI_Status_Message := 'NVRAM: Запись запрещена (STANDBY)';
        ELSE
            // Проверка на изменение данных перед записью
            L_Data_Changed := FALSE;
            FOR L_i := 0 TO VI_DataSize - 1 DO
                IF GVL_Retain.G_NVRAM_Data[VI_Offset + L_i] <> L_pData[L_i] THEN
                    L_Data_Changed := TRUE;
                    EXIT;
                END_IF;
            END_FOR;

            IF L_Data_Changed THEN
                // Безопасное копирование (WRITE)
                FOR L_i := 0 TO VI_DataSize - 1 DO
                    GVL_Retain.G_NVRAM_Data[VI_Offset + L_i] := L_pData[L_i];
                END_FOR;
                VO_HMI_Status_Message := 'NVRAM: Данные успешно сохранены в RETAIN';
            ELSE
                VO_HMI_Status_Message := 'NVRAM: Данные не изменились, запись пропущена';
            END_IF;
        END_IF;
        VO_Done := TRUE;
    END_IF;
END_IF;

IF VI_Command = 0 THEN
    VO_Done := FALSE;
END_IF;
// >>> BULK_SYNC_ANCHOR: FB_NVRAM_Manager <<<
END_FUNCTION_BLOCK

(* ---- FB_Outdoor_Lighting_Manager.st ---- *)
FUNCTION_BLOCK FB_Outdoor_Lighting_Manager
VAR_INPUT
    VI_IsActivePLC : BOOL;
    VI_Current_Scenario : E_SCENARIO_TYPE;
    VI_Security_Armed : BOOL;
    VI_Is_Night : BOOL;
    VI_Time_Of_Day_MS : UDINT;
END_VAR
VAR_IN_OUT
    VIO_Rule_Actions : ARRAY[1..GVL_CONSTANTS.C_MAX_RULES] OF ST_Rule_Action;
    VI_Motion_Sensors : ARRAY[1..GVL_CONSTANTS.C_MAX_LIGHT_ZONES] OF BOOL;
END_VAR
VAR
    L_Zone : INT;
    L_Slot : INT;
    L_Light_Index : INT;
    L_Motion_Index : INT;
    L_Socket_Index : INT;
    L_Target_Level : BYTE;
    L_Target_Socket : BOOL;
    L_Dark : BOOL;
    L_Economy : BOOL;
    L_Party : BOOL;
    L_Security : BOOL;
    L_Any_Motion : BOOL;
END_VAR

GVL_OUTDOOR_LIGHTING.G_Outdoor_Dark_Active := FALSE;
GVL_OUTDOOR_LIGHTING.G_Outdoor_Economy_Active := FALSE;
GVL_OUTDOOR_LIGHTING.G_Outdoor_Party_Active := FALSE;
GVL_OUTDOOR_LIGHTING.G_Outdoor_Security_Active := FALSE;
GVL_OUTDOOR_LIGHTING.G_Outdoor_Status_Text := 'OUTDOOR DISABLED';

FOR L_Zone := 1 TO GVL_CONSTANTS.C_MAX_OUTDOOR_ZONES DO
    GVL_OUTDOOR_LIGHTING.G_Outdoor_Light_Level[L_Zone] := 0;
    GVL_OUTDOOR_LIGHTING.G_Outdoor_Socket_State[L_Zone] := FALSE;
END_FOR;

IF (NOT VI_IsActivePLC) OR (NOT GVL_OUTDOOR_LIGHTING.G_Outdoor_Enabled) THEN
    RETURN;
END_IF;

L_Dark := FALSE;
IF GVL_OUTDOOR_LIGHTING.G_Outdoor_Fallback_To_Night THEN
    L_Dark := VI_Is_Night;
END_IF;
IF GVL_OUTDOOR_LIGHTING.G_Outdoor_Use_Lux_Sensor AND GVL_STATE.G_Ambient_Lux_Valid THEN
    L_Dark := L_Dark OR (GVL_STATE.G_Ambient_Lux < GVL_OUTDOOR_LIGHTING.G_Outdoor_Lux_Threshold);
END_IF;

IF GVL_OUTDOOR_LIGHTING.G_Outdoor_Economy_Start_MS <= GVL_OUTDOOR_LIGHTING.G_Outdoor_Economy_End_MS THEN
    L_Economy := (VI_Time_Of_Day_MS >= GVL_OUTDOOR_LIGHTING.G_Outdoor_Economy_Start_MS) AND (VI_Time_Of_Day_MS < GVL_OUTDOOR_LIGHTING.G_Outdoor_Economy_End_MS);
ELSE
    L_Economy := (VI_Time_Of_Day_MS >= GVL_OUTDOOR_LIGHTING.G_Outdoor_Economy_Start_MS) OR (VI_Time_Of_Day_MS < GVL_OUTDOOR_LIGHTING.G_Outdoor_Economy_End_MS);
END_IF;

L_Party := (VI_Current_Scenario = E_SCENARIO_TYPE.SCENARIO_PARTY);
L_Any_Motion := FALSE;
FOR L_Zone := 1 TO GVL_CONSTANTS.C_MAX_OUTDOOR_ZONES DO
    L_Motion_Index := GVL_OUTDOOR_LIGHTING.G_Outdoor_Motion_Zone_Index[L_Zone];
    IF (L_Motion_Index >= 1) AND (L_Motion_Index <= GVL_CONSTANTS.C_MAX_LIGHT_ZONES) THEN
        L_Any_Motion := L_Any_Motion OR VI_Motion_Sensors[L_Motion_Index];
    END_IF;
END_FOR;
L_Security := VI_Security_Armed AND L_Any_Motion;

GVL_OUTDOOR_LIGHTING.G_Outdoor_Dark_Active := L_Dark;
GVL_OUTDOOR_LIGHTING.G_Outdoor_Economy_Active := L_Dark AND L_Economy;
GVL_OUTDOOR_LIGHTING.G_Outdoor_Party_Active := L_Party;
GVL_OUTDOOR_LIGHTING.G_Outdoor_Security_Active := L_Security;

FOR L_Zone := 1 TO GVL_CONSTANTS.C_MAX_OUTDOOR_ZONES DO
    IF GVL_OUTDOOR_LIGHTING.G_Outdoor_Manual_Mode[L_Zone] THEN
        L_Target_Level := GVL_OUTDOOR_LIGHTING.G_Outdoor_Manual_Light_Level[L_Zone];
        L_Target_Socket := GVL_OUTDOOR_LIGHTING.G_Outdoor_Manual_Socket_State[L_Zone];
    ELSIF L_Party THEN
        L_Target_Level := GVL_OUTDOOR_LIGHTING.G_Outdoor_Party_Level;
        L_Target_Socket := GVL_OUTDOOR_LIGHTING.G_Outdoor_Sockets_Enabled AND GVL_OUTDOOR_LIGHTING.G_Outdoor_Sockets_On_In_Party;
    ELSIF L_Security THEN
        L_Target_Level := GVL_OUTDOOR_LIGHTING.G_Outdoor_Security_Level;
        L_Target_Socket := GVL_OUTDOOR_LIGHTING.G_Outdoor_Sockets_Enabled AND NOT GVL_OUTDOOR_LIGHTING.G_Outdoor_Sockets_Off_In_Security;
    ELSIF L_Dark AND L_Economy THEN
        L_Target_Level := GVL_OUTDOOR_LIGHTING.G_Outdoor_Economy_Level;
        L_Target_Socket := FALSE;
    ELSIF L_Dark THEN
        L_Target_Level := GVL_OUTDOOR_LIGHTING.G_Outdoor_Auto_Level;
        L_Target_Socket := GVL_OUTDOOR_LIGHTING.G_Outdoor_Sockets_Enabled AND GVL_OUTDOOR_LIGHTING.G_Outdoor_Sockets_On_In_Auto;
    ELSE
        L_Target_Level := 0;
        L_Target_Socket := FALSE;
    END_IF;

    GVL_OUTDOOR_LIGHTING.G_Outdoor_Light_Level[L_Zone] := L_Target_Level;
    GVL_OUTDOOR_LIGHTING.G_Outdoor_Socket_State[L_Zone] := L_Target_Socket;

    L_Light_Index := GVL_OUTDOOR_LIGHTING.G_Outdoor_Light_Zone_Index[L_Zone];
    IF (L_Light_Index >= 1) AND (L_Light_Index <= GVL_CONSTANTS.C_MAX_LIGHT_ZONES) THEN
        FOR L_Slot := 1 TO GVL_CONSTANTS.C_MAX_RULES DO
            IF NOT VIO_Rule_Actions[L_Slot].Active THEN
                VIO_Rule_Actions[L_Slot].Active := TRUE;
                VIO_Rule_Actions[L_Slot].Triggered := FALSE;
                VIO_Rule_Actions[L_Slot].Action_Type := E_Rule_Action_Type.ACTION_SET_LIGHTING_BASE;
                VIO_Rule_Actions[L_Slot].Target_ID := TO_BYTE(L_Light_Index);
                VIO_Rule_Actions[L_Slot].Value := TO_REAL(L_Target_Level);
                EXIT;
            END_IF;
        END_FOR;
    END_IF;

    L_Socket_Index := GVL_OUTDOOR_LIGHTING.G_Outdoor_Socket_Index[L_Zone];
    IF (L_Socket_Index >= 1) AND (L_Socket_Index <= GVL_CONSTANTS.C_MAX_SOCKETS) THEN
        FOR L_Slot := 1 TO GVL_CONSTANTS.C_MAX_RULES DO
            IF NOT VIO_Rule_Actions[L_Slot].Active THEN
                VIO_Rule_Actions[L_Slot].Active := TRUE;
                VIO_Rule_Actions[L_Slot].Triggered := FALSE;
                VIO_Rule_Actions[L_Slot].Action_Type := E_Rule_Action_Type.ACTION_SET_SOCKET;
                VIO_Rule_Actions[L_Slot].Target_ID := TO_BYTE(L_Socket_Index);
                IF L_Target_Socket THEN
                    VIO_Rule_Actions[L_Slot].Value := REAL#1.0;
                ELSE
                    VIO_Rule_Actions[L_Slot].Value := REAL#0.0;
                END_IF;
                EXIT;
            END_IF;
        END_FOR;
    END_IF;
END_FOR;

IF L_Party THEN
    GVL_OUTDOOR_LIGHTING.G_Outdoor_Status_Text := 'OUTDOOR PARTY';
ELSIF L_Security THEN
    GVL_OUTDOOR_LIGHTING.G_Outdoor_Status_Text := 'OUTDOOR SECURITY';
ELSIF L_Dark AND L_Economy THEN
    GVL_OUTDOOR_LIGHTING.G_Outdoor_Status_Text := 'OUTDOOR ECONOMY';
ELSIF L_Dark THEN
    GVL_OUTDOOR_LIGHTING.G_Outdoor_Status_Text := 'OUTDOOR AUTO';
ELSE
    GVL_OUTDOOR_LIGHTING.G_Outdoor_Status_Text := 'OUTDOOR DAY OFF';
END_IF;

// >>> BULK_SYNC_ANCHOR: FB_Outdoor_Lighting_Manager <<<
END_FUNCTION_BLOCK

(* ---- FB_Redundancy_Manager.st ---- *)
FUNCTION_BLOCK FB_Redundancy_Manager
VAR_INPUT
    VI_System_Time_MS : UDINT; // Системное время (мс)
    VI_Local_PLC_ID : BYTE; // 1 = ПЛК А, 2 = ПЛК B
    VI_Remote_Pulse : BOOL; // Сигнал от партнера
    VI_Remote_Is_Active : BOOL; // Статус партнера
    VI_Gateway_Ping_OK : BOOL; // Пинг до шлюза
    VI_Remote_State : ST_System_State_Snapshot; // Состояние партнера
    VI_Local_State : ST_System_State_Snapshot; // Локальное состояние
END_VAR
VAR_OUTPUT
    VO_Local_Role : E_PLC_ROLE; // Локальная роль ПЛК (Active/Standby)
    VO_Local_Pulse : BOOL; // Локальный сигнал пульса для партнера
    VO_Sync_Data_Req : BOOL; // Запрос на синхронизацию данных
    VO_Status_Msg : STRING(200); // Строковое сообщение о статусе
    VO_Synced_State : ST_System_State_Snapshot; // Синхронизированное состояние
    VO_State_Updated : BOOL; // Флаг: Состояние было обновлено
END_VAR
VAR
    L_Heartbeat : FB_PLC_Heartbeat;
    L_Pulse_Timer : FB_System_Timer;
    L_Pulse_State : BOOL;
    L_Prev_Role : E_PLC_ROLE;
    L_State_Replicator : FB_State_Replication;
END_VAR

// 1. Генерация собственного пульса (меандр 100 мс)
L_Pulse_Timer(IN := NOT L_Pulse_Timer.Q, PT := T#100ms, VI_System_Time_MS := VI_System_Time_MS);
IF L_Pulse_Timer.Q THEN
    L_Pulse_State := NOT L_Pulse_State;
END_IF;
VO_Local_Pulse := L_Pulse_State;

// 2. Определение роли через Heartbeat
L_Heartbeat(
    VI_Local_ID := VI_Local_PLC_ID,
    VI_System_Time := VI_System_Time_MS,
    VI_Remote_Pulse := VI_Remote_Pulse,
    VI_Remote_Is_Active := VI_Remote_Is_Active,
    VI_Gateway_Ping_OK := VI_Gateway_Ping_OK
);

IF L_Heartbeat.VO_Is_Active THEN
    VO_Local_Role := E_PLC_ROLE.ROLE_ACTIVE;
    VO_Status_Msg := 'ПЛК АКТИВЕН (ВЕДУЩИЙ)';
ELSE
    VO_Local_Role := E_PLC_ROLE.ROLE_STANDBY;
    VO_Status_Msg := 'ПЛК В РЕЗЕРВЕ (ВЕДОМЫЙ)';
END_IF;

// 3. Запрос на синхронизацию при переходе в ACTIVE
IF VO_Local_Role = E_PLC_ROLE.ROLE_ACTIVE AND L_Prev_Role = E_PLC_ROLE.ROLE_STANDBY THEN
    VO_Sync_Data_Req := TRUE;
ELSE
    VO_Sync_Data_Req := FALSE;
END_IF;

L_State_Replicator(
    VI_Local_Role := VO_Local_Role,
    VI_Sync_Req := VO_Sync_Data_Req,
    VI_Local_State := VI_Local_State,
    VI_Remote_State := VI_Remote_State,
    VI_System_Time_MS := VI_System_Time_MS
);
VO_Synced_State := L_State_Replicator.VO_Synced_State;
VO_State_Updated := L_State_Replicator.VO_State_Updated;

L_Prev_Role := VO_Local_Role;
// >>> BULK_SYNC_ANCHOR: FB_Redundancy_Manager <<<
END_FUNCTION_BLOCK

(* ---- FB_Runtime_Bus_Replication.st ---- *)
FUNCTION_BLOCK FB_Runtime_Bus_Replication
VAR_INPUT
    VI_Enable : BOOL;
    VI_System_Time_MS : UDINT;
END_VAR
VAR
    L_Frame : ST_Runtime_Bus_Frame;
    L_TX_Index : UINT;

    L_Finalized_Runtime_Continuity : BOOL;
END_VAR

IF NOT VI_Enable THEN
    GVL_Runtime_Bus.G_Runtime_Valid := FALSE;
    RETURN;
END_IF;

L_Finalized_Runtime_Continuity :=
    GVL_SEMANTIC_PROGRESS.Semantic_Forward_Progress_Valid
    AND GVL_SEMANTIC_PROGRESS.Semantic_Execution_Continuity_OK
    AND NOT GVL_SEMANTIC_PROGRESS.Semantic_Progress_Lease_Expired
    AND NOT GVL_SEMANTIC_PROGRESS.Semantic_Progress_Quarantine_Active
    AND GVL_RUNTIME_SNAPSHOT.Snapshot_Frozen
    AND GVL_RUNTIME_SNAPSHOT.Snapshot_Publication_Allowed
    AND GVL_RUNTIME_SNAPSHOT.Snapshot_Copy_Valid
    AND GVL_RUNTIME_SNAPSHOT.Snapshot_Isolation_Valid
    AND NOT GVL_RUNTIME_SNAPSHOT.Snapshot_Mutation_Detected
    AND GVL_DISTRIBUTED_SNAPSHOT.Distributed_Publication_Reconciled
    AND GVL_DISTRIBUTED_SNAPSHOT.Distributed_Publication_Freeze_Valid
    AND GVL_DISTRIBUTED_SNAPSHOT.Distributed_Snapshot_Consistent
    AND GVL_DISTRIBUTED_COMMIT.Distributed_Commit_Valid
    AND GVL_DISTRIBUTED_COMMIT.Publication_Prepare_Valid
    AND GVL_DISTRIBUTED_COMMIT.Publication_Commit_Confirmed
    AND NOT GVL_DISTRIBUTED_COMMIT.Peer_Commit_Mismatch
    AND NOT GVL_DISTRIBUTED_COMMIT.Commit_Lease_Expired
    AND GVL_OUTPUT_EPOCH.Output_Publication_Valid
    AND GVL_OUTPUT_EPOCH.Output_Runtime_Epoch_Valid
    AND NOT GVL_OUTPUT_EPOCH.Output_Lease_Expired
    AND NOT GVL_OUTPUT_EPOCH.Output_Forced_Safe_Decay
    AND GVL_COMMAND_VERIFY.PreOutput_Barrier_OK
    AND NOT GVL_COMMAND_VERIFY.PreOutput_Block_IO;

L_TX_Index := UDINT_TO_UINT(GVL_Runtime_Bus.G_Last_Sequence_Id + 1);

IF L_TX_Index > 128 THEN
    L_TX_Index := 1;
END_IF;

L_Frame.Frame_Valid := TRUE;

L_Frame.Frame_Time_MS := VI_System_Time_MS;
L_Frame.Frame_Id := GVL_Runtime_Bus.G_Last_Frame_Id + 1;

L_Frame.Source_Controller_Id :=
    GVL_Distributed_Runtime.G_Local_Node_State.Controller_Id;

L_Frame.Source_Runtime_Node_Id :=
    GVL_Distributed_Runtime.G_Local_Node_State.Runtime_Node_Id;

L_Frame.Frame_Sequence_Id :=
    GVL_Runtime_Bus.G_Last_Sequence_Id + 1;

L_Frame.Frame_Ack_Required := TRUE;

L_Frame.Authority_State_Frame := TRUE;
L_Frame.Recovery_State_Frame := TRUE;
L_Frame.Quarantine_State_Frame := TRUE;
L_Frame.Topology_State_Frame := TRUE;
L_Frame.Binding_State_Frame := TRUE;
L_Frame.Predictive_State_Frame := TRUE;

IF GVL_Distributed_Authority.G_Distributed_Safety_Barrier_OK
   AND NOT GVL_Distributed_Runtime.G_Split_Brain_Suspected
   AND L_Finalized_Runtime_Continuity THEN

    L_Frame.Replication_Consistent := TRUE;

    L_Frame.Status_Code := 0;
    L_Frame.Status_Text :=
        'Deterministic replication frame accepted';

ELSE

    L_Frame.Replication_Rejected := TRUE;

    L_Frame.Status_Code := 2;
    L_Frame.Status_Text :=
        'Deterministic replication frame rejected';

END_IF;

GVL_Runtime_Bus.G_TX_Frames[L_TX_Index] := L_Frame;

GVL_Runtime_Bus.G_Last_Frame_Id :=
    L_Frame.Frame_Id;

GVL_Runtime_Bus.G_Last_Sequence_Id :=
    L_Frame.Frame_Sequence_Id;

GVL_Runtime_Bus.G_TX_Healthy :=
    L_Frame.Replication_Consistent;

GVL_Runtime_Bus.G_RX_Healthy := TRUE;

GVL_Runtime_Bus.G_Any_Replication_Rejected :=
    L_Frame.Replication_Rejected;

GVL_Runtime_Bus.G_Runtime_Valid := TRUE;
GVL_Runtime_Bus.G_Last_Update_MS := VI_System_Time_MS;

IF L_Frame.Replication_Rejected THEN
    GVL_Runtime_Bus.G_Status_Code := 2;
    GVL_Runtime_Bus.G_Status_Text :=
        'Runtime bus replication rejected';
ELSE
    GVL_Runtime_Bus.G_Status_Code := 0;
    GVL_Runtime_Bus.G_Status_Text :=
        'Runtime bus replication healthy';
END_IF;

END_FUNCTION_BLOCK

(* ---- FB_Runtime_Node_Discovery.st ---- *)
FUNCTION_BLOCK FB_Runtime_Node_Discovery
VAR_INPUT
    VI_Enable : BOOL;
    VI_System_Time_MS : UDINT;
END_VAR
VAR
    L_i : INT;
    L_State : ST_Runtime_Node_Discovery_State;

    L_Any_Quarantine : BOOL;
    L_Any_Rejected : BOOL;

    L_Finalized_Runtime_Continuity : BOOL;
END_VAR

IF NOT VI_Enable THEN
    GVL_Runtime_Discovery.G_Runtime_Valid := FALSE;
    RETURN;
END_IF;

// Finalized runtime continuity proof chain.
L_Finalized_Runtime_Continuity :=
    GVL_SEMANTIC_PROGRESS.Semantic_Forward_Progress_Valid
    AND GVL_SEMANTIC_PROGRESS.Semantic_Execution_Continuity_OK
    AND NOT GVL_SEMANTIC_PROGRESS.Semantic_Progress_Lease_Expired
    AND NOT GVL_SEMANTIC_PROGRESS.Semantic_Progress_Quarantine_Active
    AND GVL_RUNTIME_SNAPSHOT.Snapshot_Frozen
    AND GVL_RUNTIME_SNAPSHOT.Snapshot_Publication_Allowed
    AND GVL_RUNTIME_SNAPSHOT.Snapshot_Copy_Valid
    AND GVL_RUNTIME_SNAPSHOT.Snapshot_Isolation_Valid
    AND NOT GVL_RUNTIME_SNAPSHOT.Snapshot_Mutation_Detected
    AND GVL_DISTRIBUTED_SNAPSHOT.Distributed_Publication_Reconciled
    AND GVL_DISTRIBUTED_SNAPSHOT.Distributed_Publication_Freeze_Valid
    AND GVL_DISTRIBUTED_SNAPSHOT.Distributed_Snapshot_Consistent
    AND GVL_DISTRIBUTED_COMMIT.Distributed_Commit_Valid
    AND GVL_DISTRIBUTED_COMMIT.Publication_Prepare_Valid
    AND GVL_DISTRIBUTED_COMMIT.Publication_Commit_Confirmed
    AND NOT GVL_DISTRIBUTED_COMMIT.Peer_Commit_Mismatch
    AND NOT GVL_DISTRIBUTED_COMMIT.Commit_Lease_Expired
    AND GVL_OUTPUT_EPOCH.Output_Publication_Valid
    AND GVL_OUTPUT_EPOCH.Output_Runtime_Epoch_Valid
    AND NOT GVL_OUTPUT_EPOCH.Output_Lease_Expired
    AND NOT GVL_OUTPUT_EPOCH.Output_Forced_Safe_Decay
    AND GVL_COMMAND_VERIFY.PreOutput_Barrier_OK
    AND NOT GVL_COMMAND_VERIFY.PreOutput_Block_IO;

FOR L_i := 1 TO 32 DO

    L_State := GVL_Runtime_Discovery.G_Discovery_State[L_i];

    IF L_State.Discovery_Active THEN

        L_State.Runtime_Valid := TRUE;
        L_State.Runtime_System_Time_MS := VI_System_Time_MS;

        L_State.Node_Discovered := TRUE;

        IF GVL_Distributed_Authority.G_Distributed_Safety_Barrier_OK
           AND NOT GVL_Runtime_Sessions.G_Any_Stale_Session
           AND L_Finalized_Runtime_Continuity THEN

            L_State.Node_Validated := TRUE;
            L_State.Node_Authorized := TRUE;

            L_State.Capability_Validated := TRUE;
            L_State.Execution_Domain_Assigned := TRUE;
            L_State.Deployment_Assigned := TRUE;

            L_State.Status_Code := 0;
            L_State.Status_Text :=
                'Runtime node discovery healthy';

        ELSE

            L_State.Node_Quarantined := TRUE;
            L_State.Discovery_Rejected := TRUE;

            L_Any_Quarantine := TRUE;
            L_Any_Rejected := TRUE;

            L_State.Status_Code := 2;
            L_State.Status_Text :=
                'Runtime node discovery rejected';

        END_IF;

        GVL_Runtime_Discovery.G_Discovery_State[L_i] :=
            L_State;

    END_IF;

END_FOR;

GVL_Runtime_Discovery.G_Any_Node_Quarantined :=
    L_Any_Quarantine;

GVL_Runtime_Discovery.G_Any_Discovery_Rejected :=
    L_Any_Rejected;

GVL_Runtime_Discovery.G_Runtime_Valid := TRUE;
GVL_Runtime_Discovery.G_Last_Update_MS := VI_System_Time_MS;

IF L_Any_Rejected THEN
    GVL_Runtime_Discovery.G_Status_Code := 2;
    GVL_Runtime_Discovery.G_Status_Text :=
        'Runtime discovery rejection detected';
ELSIF L_Any_Quarantine THEN
    GVL_Runtime_Discovery.G_Status_Code := 1;
    GVL_Runtime_Discovery.G_Status_Text :=
        'Runtime discovery quarantine active';
ELSE
    GVL_Runtime_Discovery.G_Status_Code := 0;
    GVL_Runtime_Discovery.G_Status_Text :=
        'Runtime discovery governance healthy';
END_IF;

END_FUNCTION_BLOCK

(* ---- FB_Safety_Manager.st ---- *)
FUNCTION_BLOCK FB_Safety_Manager
VAR_INPUT
    VI_Gas_Alarm : BOOL;
    VI_Leak_Alarm : BOOL;
    VI_Smoke_Alarm : BOOL;
    VI_Reset : BOOL; // Ручной сброс защёлкнутых safety-аварий оператором
END_VAR
VAR_OUTPUT
    VO_Gas_Latched : BOOL;
    VO_Leak_Latched : BOOL;
    VO_Smoke_Latched : BOOL;
    VO_Emergency_Stop : BOOL;
END_VAR
VAR
    L_Any_Active : BOOL;
END_VAR

// Защёлкиваем аварии независимо друг от друга
IF VI_Gas_Alarm THEN
    VO_Gas_Latched := TRUE;
END_IF;

IF VI_Leak_Alarm THEN
    VO_Leak_Latched := TRUE;
END_IF;

IF VI_Smoke_Alarm THEN
    VO_Smoke_Latched := TRUE;
END_IF;

L_Any_Active := VI_Gas_Alarm OR VI_Leak_Alarm OR VI_Smoke_Alarm;

// Ручной сброс допустим только когда все входные аварийные сигналы уже исчезли
IF VI_Reset AND NOT L_Any_Active THEN
    VO_Gas_Latched := FALSE;
    VO_Leak_Latched := FALSE;
    VO_Smoke_Latched := FALSE;
END_IF;

// Агрегированный аварийный стоп = любая защёлкнутая safety-авария
VO_Emergency_Stop := VO_Gas_Latched OR VO_Leak_Latched OR VO_Smoke_Latched;
END_FUNCTION_BLOCK
// >>> BULK_SYNC_ANCHOR: FB_Safety_Manager <<<

(* ---- FB_Scenario_Transition_Controller.st ---- *)
FUNCTION_BLOCK FB_Scenario_Transition_Controller
VAR_INPUT
    VI_System_Time : UDINT;
    VI_Start_Time  : UDINT;
    VI_Duration    : UDINT; // Длительность перехода (мс)
    VI_Start_Value : REAL;  // Начальное значение
    VI_End_Value   : REAL;  // Конечное значение
END_VAR
VAR_OUTPUT
    VO_Current_Value : REAL; // Текущее интерполированное значение
    VO_Transition_Done : BOOL; // Флаг завершения перехода
END_VAR
VAR
    L_Elapsed : UDINT;
    L_Progress : REAL;
END_VAR

L_Elapsed := (SEL(VI_System_Time >= VI_Start_Time, VI_System_Time - VI_Start_Time, (4294967295 - VI_Start_Time) + VI_System_Time + 1));

IF L_Elapsed >= VI_Duration OR VI_Duration = 0 THEN
    VO_Current_Value := VI_End_Value;
    VO_Transition_Done := TRUE;
ELSE
    L_Progress := UDINT_TO_REAL(L_Elapsed) / UDINT_TO_REAL(VI_Duration);
    VO_Current_Value := VI_Start_Value + (VI_End_Value - VI_Start_Value) * L_Progress;
    VO_Transition_Done := FALSE;
END_IF;
END_FUNCTION_BLOCK

(* ---- FB_Sensor_Calibration_Processor.st ---- *)
FUNCTION_BLOCK FB_Sensor_Calibration_Processor
VAR_INPUT
    VI_Raw_Value : REAL;
    VI_Record    : ST_Sensor_Calibration_Record;
END_VAR
VAR_OUTPUT
    VO_Calibrated_Value : REAL;
    VO_Record_Valid : BOOL;
    VO_Calibration_Applied : BOOL;
    VO_Record_Fault : BOOL;
    VO_Used_Offset : REAL;
    VO_Used_Multiplier : REAL;
    VO_Last_Calibration_Timestamp : UDINT;
END_VAR
VAR
    L_Record_Has_Correction : BOOL;
    L_Multiplier_In_Range : BOOL;
END_VAR

// Calibration records are allowed to be neutral by default:
// multiplier=1.0, offset=0.0, verification_passed=FALSE.
// Non-neutral corrections must be verified before they affect normalized IO.
L_Record_Has_Correction := (VI_Record.offset <> 0.0) OR (VI_Record.multiplier <> 1.0);
L_Multiplier_In_Range := (VI_Record.multiplier >= 0.01) AND (VI_Record.multiplier <= 100.0);

VO_Record_Valid := TRUE;
VO_Record_Fault := FALSE;
VO_Calibration_Applied := FALSE;
VO_Used_Offset := 0.0;
VO_Used_Multiplier := 1.0;
VO_Last_Calibration_Timestamp := VI_Record.last_calibration_timestamp;

IF NOT L_Multiplier_In_Range THEN
    VO_Record_Valid := FALSE;
    VO_Record_Fault := TRUE;
ELSIF L_Record_Has_Correction AND NOT VI_Record.verification_passed THEN
    VO_Record_Valid := FALSE;
    VO_Record_Fault := TRUE;
END_IF;

IF VO_Record_Valid THEN
    VO_Used_Offset := VI_Record.offset;
    VO_Used_Multiplier := VI_Record.multiplier;
    VO_Calibration_Applied := L_Record_Has_Correction OR (VI_Record.last_calibration_timestamp <> 0);
    VO_Calibrated_Value := (VI_Raw_Value * VI_Record.multiplier) + VI_Record.offset;
ELSE
    // Fail safe for invalid calibration records: publish raw normalized input
    // and let the caller raise diagnostics through VO_Record_Fault.
    VO_Calibrated_Value := VI_Raw_Value;
END_IF;
END_FUNCTION_BLOCK

(* ---- FB_State_Manager.st ---- *)
FUNCTION_BLOCK FB_State_Manager
VAR_INPUT
    VI_System_Severity : E_System_Severity;
    VI_Root_Cause      : E_System_Root_Cause;
    VI_Freeze_Risk     : BOOL := FALSE;
END_VAR

VAR_OUTPUT
    VO_System_OK        : BOOL;
    VO_System_Warning   : BOOL;
    VO_System_Critical  : BOOL;
    VO_Status_Msg       : STRING(200);

    // compatibility output for existing orchestration
    VO_System_Mode      : E_System_Operating_Mode;
END_VAR

VAR
    L_Requested_Mode : E_System_Operating_Mode;
END_VAR

VO_System_OK := FALSE;
VO_System_Warning := FALSE;
VO_System_Critical := FALSE;
VO_Status_Msg := '';

// ------------------------------------------------------
// Stateful deterministic mode governance.
// ------------------------------------------------------
// SAFE_STOP entry is immediate.
// SAFE_STOP exit is convergence-lease gated.
//
// Prevents one-cycle false recovery and transient
// healthy visibility from restoring system operation.
// ------------------------------------------------------

L_Requested_Mode := E_System_Operating_Mode.MODE_NORMAL;

CASE VI_System_Severity OF
    E_System_Severity.SEV_NORMAL:
        VO_System_OK := TRUE;
        VO_Status_Msg := 'Система в норме';
        L_Requested_Mode := E_System_Operating_Mode.MODE_NORMAL;

    E_System_Severity.SEV_WARNING:
        VO_System_Warning := TRUE;
        L_Requested_Mode := E_System_Operating_Mode.MODE_DEGRADED;

        CASE VI_Root_Cause OF
            E_System_Root_Cause.ROOT_WATER_LEAK:
                VO_Status_Msg := 'Предупреждение: протечка воды';

            E_System_Root_Cause.ROOT_CO_WARNING:
                VO_Status_Msg := 'Предупреждение: повышенный CO';

            ELSE
                VO_Status_Msg := 'Предупреждение системы';
        END_CASE;

    E_System_Severity.SEV_DEGRADED:
        VO_System_Warning := TRUE;
        L_Requested_Mode := E_System_Operating_Mode.MODE_DEGRADED;

        CASE VI_Root_Cause OF
            E_System_Root_Cause.ROOT_SENSOR_FAULT:
                VO_Status_Msg := 'Деградация: ошибка датчика';

            E_System_Root_Cause.ROOT_IO_OFFLINE:
                VO_Status_Msg := 'Деградация: модуль IO недоступен';

            E_System_Root_Cause.ROOT_COMM_FAULT:
                VO_Status_Msg := 'Деградация: ошибка связи';

            E_System_Root_Cause.ROOT_WATCHDOG_FAULT:
                VO_Status_Msg := 'Деградация: watchdog fault';

            E_System_Root_Cause.ROOT_SUBSYSTEM_FAULT:
                VO_Status_Msg := 'Деградация: ошибка подсистемы';

            ELSE
                VO_Status_Msg := 'Деградация системы';
        END_CASE;

    E_System_Severity.SEV_CRITICAL:
        VO_System_Critical := TRUE;

        IF (VI_Root_Cause = E_System_Root_Cause.ROOT_GAS_LEAK OR
            VI_Root_Cause = E_System_Root_Cause.ROOT_CO_CRITICAL) AND
            VI_Freeze_Risk THEN
            L_Requested_Mode := E_System_Operating_Mode.MODE_FREEZE_PROTECTION;
        ELSE
            L_Requested_Mode := E_System_Operating_Mode.MODE_SAFE_STOP;
        END_IF;

        CASE VI_Root_Cause OF
            E_System_Root_Cause.ROOT_FIRE:
                VO_Status_Msg := 'АВАРИЯ: ПОЖАР';

            E_System_Root_Cause.ROOT_GAS_LEAK:
                VO_Status_Msg := 'АВАРИЯ: УТЕЧКА ГАЗА';

            E_System_Root_Cause.ROOT_CO_CRITICAL:
                VO_Status_Msg := 'АВАРИЯ: КРИТИЧЕСКИЙ CO';

            E_System_Root_Cause.ROOT_WATCHDOG_FAULT:
                VO_Status_Msg := 'АВАРИЯ: WATCHDOG';

            ELSE
                VO_Status_Msg := 'АВАРИЯ СИСТЕМЫ';
        END_CASE;
END_CASE;

// ------------------------------------------------------
// Deterministic SAFE_STOP exit hardening.
// ------------------------------------------------------
// SAFE_STOP/FREEZE_PROTECTION exit requires sustained
// convergence evidence and convergence lease acquisition.
// ------------------------------------------------------

IF (VO_System_Mode = E_System_Operating_Mode.MODE_SAFE_STOP)
OR (VO_System_Mode = E_System_Operating_Mode.MODE_FREEZE_PROTECTION)
THEN
    IF (L_Requested_Mode <> E_System_Operating_Mode.MODE_SAFE_STOP)
    AND (L_Requested_Mode <> E_System_Operating_Mode.MODE_FREEZE_PROTECTION)
    THEN
        IF NOT GVL_CONVERGENCE.Convergence_Lease_OK THEN
            // Hold previous safe mode until deterministic
            // convergence/recovery proof exists.
            L_Requested_Mode := VO_System_Mode;

            IF VO_Status_Msg = '' THEN
                VO_Status_Msg := 'Ожидание подтверждения восстановления';
            ELSE
                VO_Status_Msg := CONCAT(VO_Status_Msg, ' | convergence pending');
            END_IF;
        END_IF;
    END_IF;
END_IF;

VO_System_Mode := L_Requested_Mode;

// >>> BULK_SYNC_ANCHOR: FB_State_Manager <<<
END_FUNCTION_BLOCK

(* ---- FB_State_Trace_Log.st ---- *)
FUNCTION_BLOCK FB_State_Trace_Log
VAR_INPUT
    VI_System_Time : UDINT;
    VI_Gas_Alarm : BOOL;
    VI_Leak_Alarm : BOOL;
    VI_Pumps : ARRAY[1..4] OF BOOL;
END_VAR
VAR_OUTPUT
    VO_Last_Change_Time : UDINT;
END_VAR
VAR
    L_i : INT;
    L_Last_Gas : BOOL;
    L_Last_Leak : BOOL;
    L_Last_Pumps : ARRAY[1..4] OF BOOL;
    L_Changed : BOOL;
END_VAR

L_Changed :=
    (VI_Gas_Alarm <> L_Last_Gas)
    OR (VI_Leak_Alarm <> L_Last_Leak);

FOR L_i := 1 TO 4 DO
    IF VI_Pumps[L_i] <> L_Last_Pumps[L_i] THEN
        L_Changed := TRUE;
    END_IF;
END_FOR;

IF L_Changed THEN
    VO_Last_Change_Time := VI_System_Time;
END_IF;

L_Last_Gas := VI_Gas_Alarm;
L_Last_Leak := VI_Leak_Alarm;

FOR L_i := 1 TO 4 DO
    L_Last_Pumps[L_i] := VI_Pumps[L_i];
END_FOR;

END_FUNCTION_BLOCK

(* ---- FB_System_Diagnostics.st ---- *)
// ==============================================================================
// System diagnostics helper
//
// Legacy compatibility helper.
//
// IMPORTANT:
// This function block must not write aggregated diagnostics fields directly.
// Aggregated diagnostics ownership is centralized in:
//
//   FB_System_Health_Orchestrator
//
// Protected aggregate fields:
//
//   GVL_STATUS.G_Diagnostics.Sensor_Fault
//   GVL_STATUS.G_Diagnostics.IO_Offline
//   GVL_STATUS.G_Diagnostics.Subsystem_Degraded
//
// This stub is intentionally side-effect free to prevent resurrecting duplicate
// diagnostics aggregate writers from legacy call paths.
// ==============================================================================
FUNCTION_BLOCK FB_System_Diagnostics

// Intentionally side-effect free.
// Diagnostics aggregate projection is owned by FB_System_Health_Orchestrator.

// >>> BULK_SYNC_ANCHOR: FB_System_Diagnostics <<<
END_FUNCTION_BLOCK

(* ---- FB_System_Redundancy_Orchestrator.st ---- *)
// ==============================================================================
// System redundancy orchestrator helper
//
// Cold-spare architecture helper. The active runtime is local-only; a second PLC
// is not allowed to hot-apply replicated state or arbitrate the same physical
// outputs. This block only builds the local snapshot for diagnostics/future
// backup use and publishes local service status.
// ==============================================================================
FUNCTION_BLOCK FB_System_Redundancy_Orchestrator
VAR_IN_OUT
    VIO_Local_State : ST_System_State_Snapshot;
    VIO_Remote_State : ST_System_State_Snapshot;
END_VAR

// Build local state snapshot for diagnostics / future backup export.
VIO_Local_State.System_Time_MS := GVL_STATUS.G_System_Time_MS;
VIO_Local_State.Current_Scenario := GVL_STATUS.G_Current_Scenario;
VIO_Local_State.Security_Armed := GVL_ALARM.G_Security_Armed;
VIO_Local_State.Active_Alarms := GVL_ALARM.G_Active_Alarm_Count;
VIO_Local_State.Zone_Valves := GVL_STATE.G_Zone_Valves;
VIO_Local_State.Manifold_Pumps := GVL_STATE.G_Manifold_Pumps;
VIO_Local_State.Lighting_States := GVL_STATE.G_Lighting_Levels;
VIO_Local_State.Blinds_Positions := GVL_STATE.G_Blinds_Positions;
VIO_Local_State.Socket_States := GVL_STATE.G_Socket_States;
VIO_Local_State.Gas_Valve_Closed := GVL_COMMAND.G_Gas_Valve_Close;
VIO_Local_State.Water_Valves_Closed := GVL_COMMAND.G_Close_Valve_36;
VIO_Local_State.Version := VIO_Local_State.Version + 1;

// Local-only role projection. No remote-state apply is permitted here.
GVL_STATUS.G_Is_Active_PLC := TRUE;
GVL_STATUS.G_Other_PLC_Is_Active := FALSE;
GVL_IO.DO_Active_Status := TRUE;

// Keep the remote snapshot untouched; it is intentionally not applied to any
// status/alarm/state/command GVL in cold-spare mode.

// >>> BULK_SYNC_ANCHOR: FB_System_Redundancy_Orchestrator <<<
END_FUNCTION_BLOCK

(* ---- FB_System_Timer.st ---- *)
// ==============================================================================
// Блок таймера, привязанный к системному времени (System Timer)
// Назначение:
// - Замена стандартного TON для обеспечения точной выдержки времени,
//   независимой от времени цикла ПЛК, с использованием единого системного времени.
// ==============================================================================
FUNCTION_BLOCK FB_System_Timer
VAR_INPUT
    IN : BOOL; // Вход запуска таймера
    PT : TIME; // Заданное время
    VI_System_Time_MS : UDINT; // Системное время (мс)
END_VAR
VAR_OUTPUT
    Q : BOOL; // Выход: таймер сработал
    ET : TIME; // Прошедшее время
END_VAR
VAR
    L_Start_Time : UDINT;
    L_Running : BOOL;
END_VAR

IF IN THEN
    IF NOT L_Running THEN
        L_Start_Time := VI_System_Time_MS;
        L_Running := TRUE;
        ET := T#0s;
        Q := FALSE;
    ELSE
        // Обработка переполнения UDINT (примерно 49 дней)
        ET := TO_TIME((SEL(VI_System_Time_MS >= L_Start_Time, VI_System_Time_MS - L_Start_Time, (4294967295 - L_Start_Time) + VI_System_Time_MS + 1)));

        IF ET >= PT THEN
            Q := TRUE;
            ET := PT;
        ELSE
            Q := FALSE;
        END_IF;
    END_IF;
ELSE
    L_Running := FALSE;
    ET := T#0s;
    Q := FALSE;
END_IF;
// >>> BULK_SYNC_ANCHOR: FB_System_Timer <<<
END_FUNCTION_BLOCK

(* ---- FB_Trace_Write.st ---- *)
FUNCTION_BLOCK FB_Trace_Write
VAR_INPUT
    iLayer : E_Trace_Layer;
    iSource : E_Trace_Source;
    iReason : E_System_Reason_Code;
    iValueBool : BOOL;
    iValueReal : REAL;
    iText : STRING(120);
END_VAR

VAR
    L_Index : INT;
END_VAR

IF NOT GVL_TRACE.G_Trace_Enabled THEN RETURN; END_IF;

L_Index := GVL_TRACE.G_Trace_Write_Index;

GVL_TRACE.G_Trace_Buffer[L_Index].Timestamp_MS := GVL_TIME_SERVICE.G_Now_MS;
GVL_TRACE.G_Trace_Buffer[L_Index].Layer := iLayer;
GVL_TRACE.G_Trace_Buffer[L_Index].Source := iSource;
GVL_TRACE.G_Trace_Buffer[L_Index].Reason_Code := iReason;
GVL_TRACE.G_Trace_Buffer[L_Index].Value_Bool := iValueBool;
GVL_TRACE.G_Trace_Buffer[L_Index].Value_Real := iValueReal;
GVL_TRACE.G_Trace_Buffer[L_Index].Text := iText;

L_Index := L_Index + 1;
IF L_Index > 200 THEN L_Index := 1; END_IF;

GVL_TRACE.G_Trace_Write_Index := L_Index;
END_FUNCTION_BLOCK

(* ---- FB_Trend_Logger.st ---- *)
FUNCTION_BLOCK FB_Trend_Logger
VAR_INPUT
    VI_System_Time_MS : UDINT;
    VI_Config : ST_Trend_Config;
    VI_Current_Value : REAL;
END_VAR
VAR_OUTPUT
    VO_Data : ST_Trend_Data;
END_VAR
VAR
    L_Last_Log_Time : UDINT;
    L_Last_Value : REAL;
    L_Deviation : REAL;
    L_Elapsed_Time : UDINT;
    L_Write_Index : UDINT;
END_VAR

IF NOT VI_Config.enabled THEN
    RETURN;
END_IF;

L_Deviation := ABS(VI_Current_Value - L_Last_Value);

IF VI_System_Time_MS >= L_Last_Log_Time THEN
    L_Elapsed_Time := VI_System_Time_MS - L_Last_Log_Time;
ELSE
    L_Elapsed_Time := (4294967295 - L_Last_Log_Time) + VI_System_Time_MS + 1;
END_IF;

IF (L_Deviation >= (ABS(L_Last_Value) * VI_Config.deviation_threshold_percent / REAL#100.0)) OR
   (L_Elapsed_Time >= GVL_CONSTANTS.C_MS_IN_HOUR) THEN
    L_Write_Index := (VO_Data.record_count MOD 100) + 1;
    VO_Data.write_index := L_Write_Index;
    VO_Data.values[L_Write_Index] := VI_Current_Value;
    VO_Data.timestamps[L_Write_Index] := VI_System_Time_MS;
    VO_Data.record_count := VO_Data.record_count + 1;
    VO_Data.sum_values := VO_Data.sum_values + VI_Current_Value;
    VO_Data.config := VI_Config;
    L_Last_Value := VI_Current_Value;
    L_Last_Log_Time := VI_System_Time_MS;
END_IF;

END_FUNCTION_BLOCK

(* ---- FB_TwoFactor_Auth.st ---- *)
FUNCTION_BLOCK FB_TwoFactor_Auth
VAR_INPUT
    VI_System_Time_MS : UDINT;
    VI_Start_Auth     : BOOL;
    VI_Method         : E_TwoFactor_Method;
    VI_User_Code      : STRING(6);
    VI_Reset_Success  : BOOL; // Сброс успешного состояния
END_VAR
VAR_OUTPUT
    VO_State          : ST_TwoFactor_Auth_State;
    VO_Send_Code_Req  : BOOL; // Запрос на отправку кода (например, через шлюз)
    VO_Code_To_Send   : STRING(6); // Сгенерированный код для отправки
END_VAR
VAR
    L_Generated_Code  : STRING(6) := '';
    L_Start_Time      : UDINT;
    R_Trig_Start      : R_TRIG;
    L_Prev_User_Code  : STRING(6);
    L_Lockout_Start_Time : UDINT; // Время начала блокировки
    fbHMAC            : FB_HMAC_SHA1;
    L_Elapsed_Time    : UDINT;
    L_Time_Step       : UDINT;
    L_Message         : ARRAY[0..7] OF BYTE;
    L_Key             : ARRAY[0..63] OF BYTE;
    L_Offset          : INT;
    L_Truncated_Hash  : UDINT;
    L_i               : INT;
    L_Current_TOTP    : STRING(6);
    L_Prev_TOTP       : STRING(6);
    L_Code_Valid      : BOOL;
END_VAR

R_Trig_Start(CLK := VI_Start_Auth);

IF VI_Reset_Success THEN
    VO_State.Is_Success := FALSE;
END_IF;

IF R_Trig_Start.Q AND NOT VO_State.is_pending AND NOT VO_State.Is_Locked THEN
    VO_State.is_pending := TRUE;
    VO_State.Auth_Method := VI_Method;
    L_Start_Time := VI_System_Time_MS;
    VO_State.Attempts_Left := 3;
    VO_State.Is_Success := FALSE;
    VO_State.Is_Locked := FALSE;
    L_Prev_User_Code := '';

    IF VI_Method <> E_TwoFactor_Method.TF_METHOD_TOTP THEN
        // Генерируем одноразовый код через HMAC (без упрощенного алгоритма "по времени")
        L_Time_Step := VI_System_Time_MS / 30000;
        L_Key[0] := 16#31; L_Key[1] := 16#32; L_Key[2] := 16#33; L_Key[3] := 16#34; // Секрет-шаблон, заменяется из конфигурации
        FOR L_i := 0 TO 7 DO L_Message[7 - L_i] := TO_BYTE(SHR(L_Time_Step + L_Start_Time, L_i * 8) AND 16#FF); END_FOR;
        fbHMAC(Key := L_Key, KeyLength := 4, Message := L_Message, MessageLength := 8);
        L_Offset := TO_INT(fbHMAC.Hash[19] AND 16#0F);
        L_Truncated_Hash := (SHL(TO_UDINT(fbHMAC.Hash[L_Offset] AND 16#7F), 24) OR SHL(TO_UDINT(fbHMAC.Hash[L_Offset+1] AND 16#FF), 16) OR SHL(TO_UDINT(fbHMAC.Hash[L_Offset+2] AND 16#FF), 8) OR TO_UDINT(fbHMAC.Hash[L_Offset+3] AND 16#FF));
        L_Generated_Code := UDINT_TO_STRING(L_Truncated_Hash MOD 1000000);
        WHILE LEN(L_Generated_Code) < 6 DO
            L_Generated_Code := CONCAT('0', L_Generated_Code);
        END_WHILE;

        VO_Code_To_Send := L_Generated_Code;
        VO_Send_Code_Req := TRUE;
    ELSE
        // Для TOTP код не отправляем
        VO_Code_To_Send := '';
        VO_Send_Code_Req := FALSE;
    END_IF;
ELSE
    VO_Send_Code_Req := FALSE;
END_IF;

IF VO_State.is_pending THEN
    L_Elapsed_Time := (SEL(VI_System_Time_MS >= L_Start_Time, VI_System_Time_MS - L_Start_Time, (4294967295 - L_Start_Time) + VI_System_Time_MS + 1));

    IF L_Elapsed_Time < (GVL_CONSTANTS.C_MS_IN_MINUTE * 5) THEN
        VO_State.Time_Left_S := TO_UINT(((GVL_CONSTANTS.C_MS_IN_MINUTE * 5) - L_Elapsed_Time) / 1000);
    ELSE
        VO_State.Time_Left_S := 0;
    END_IF;

    IF VI_User_Code <> '' AND VI_User_Code <> L_Prev_User_Code THEN
        L_Code_Valid := FALSE;

        IF VI_Method = E_TwoFactor_Method.TF_METHOD_TOTP THEN
            // Вычисляем TOTP для текущего шага времени (30 секунд)
            L_Time_Step := VI_System_Time_MS / 30000;

            // Подготовка ключа (в реальном проекте берется из GVL_CONFIG)
            L_Key[0] := 16#31; L_Key[1] := 16#32; L_Key[2] := 16#33; L_Key[3] := 16#34; // '1234'

            // Проверка текущего шага
            FOR L_i := 0 TO 7 DO L_Message[7 - L_i] := TO_BYTE(SHR(L_Time_Step, L_i * 8) AND 16#FF); END_FOR;
            fbHMAC(Key := L_Key, KeyLength := 4, Message := L_Message, MessageLength := 8);
            L_Offset := TO_INT(fbHMAC.Hash[19] AND 16#0F);
            L_Truncated_Hash := (SHL(TO_UDINT(fbHMAC.Hash[L_Offset] AND 16#7F), 24) OR SHL(TO_UDINT(fbHMAC.Hash[L_Offset+1] AND 16#FF), 16) OR SHL(TO_UDINT(fbHMAC.Hash[L_Offset+2] AND 16#FF), 8) OR TO_UDINT(fbHMAC.Hash[L_Offset+3] AND 16#FF));
            L_Current_TOTP := UDINT_TO_STRING(L_Truncated_Hash MOD 1000000);
            WHILE LEN(L_Current_TOTP) < 6 DO L_Current_TOTP := CONCAT('0', L_Current_TOTP); END_WHILE;

            // Проверка предыдущего шага (для компенсации рассинхронизации)
            FOR L_i := 0 TO 7 DO L_Message[7 - L_i] := TO_BYTE(SHR(L_Time_Step - 1, L_i * 8) AND 16#FF); END_FOR;
            fbHMAC(Key := L_Key, KeyLength := 4, Message := L_Message, MessageLength := 8);
            L_Offset := TO_INT(fbHMAC.Hash[19] AND 16#0F);
            L_Truncated_Hash := (SHL(TO_UDINT(fbHMAC.Hash[L_Offset] AND 16#7F), 24) OR SHL(TO_UDINT(fbHMAC.Hash[L_Offset+1] AND 16#FF), 16) OR SHL(TO_UDINT(fbHMAC.Hash[L_Offset+2] AND 16#FF), 8) OR TO_UDINT(fbHMAC.Hash[L_Offset+3] AND 16#FF));
            L_Prev_TOTP := UDINT_TO_STRING(L_Truncated_Hash MOD 1000000);
            WHILE LEN(L_Prev_TOTP) < 6 DO L_Prev_TOTP := CONCAT('0', L_Prev_TOTP); END_WHILE;

            IF VI_User_Code = L_Current_TOTP OR VI_User_Code = L_Prev_TOTP THEN
                L_Code_Valid := TRUE;
            END_IF;
        ELSE
            IF VI_User_Code = L_Generated_Code THEN
                L_Code_Valid := TRUE;
            END_IF;
        END_IF;

        IF L_Code_Valid THEN
            VO_State.Is_Success := TRUE;
            VO_State.is_pending := FALSE;
        ELSE
            IF VO_State.Attempts_Left > 0 THEN
                VO_State.Attempts_Left := VO_State.Attempts_Left - 1;
            END_IF;

            IF VO_State.Attempts_Left = 0 THEN
                VO_State.Is_Locked := TRUE;
                VO_State.is_pending := FALSE;
                L_Lockout_Start_Time := VI_System_Time_MS; // Блокировка на 5 минут
            END_IF;
        END_IF;
    END_IF;
    L_Prev_User_Code := VI_User_Code;

    IF L_Elapsed_Time > (GVL_CONSTANTS.C_MS_IN_MINUTE * 5) THEN
        VO_State.is_pending := FALSE; // Таймаут
    END_IF;
END_IF;

IF VO_State.Is_Locked THEN
    IF (SEL(VI_System_Time_MS >= L_Lockout_Start_Time, VI_System_Time_MS - L_Lockout_Start_Time, (4294967295 - L_Lockout_Start_Time) + VI_System_Time_MS + 1)) >= (GVL_CONSTANTS.C_MS_IN_MINUTE * 5) THEN
        VO_State.Is_Locked := FALSE;
    END_IF;
END_IF;
END_FUNCTION_BLOCK

(* ---- FB_Water_Output_Projection.st ---- *)
FUNCTION_BLOCK FB_Water_Output_Projection
VAR_INPUT
    VI_Zone_Enable : ARRAY[1..GVL_CONSTANTS.C_MAX_WATER_ZONES] OF BOOL;

    // Common inlet valves: 35 = ХВС, 36 = ГВС.
    VI_Valve_35_Open : BOOL;
    VI_Valve_35_Close : BOOL;
    VI_Valve_36_Open : BOOL;
    VI_Valve_36_Close : BOOL;

    // Local riser valves: 1/2 riser 1, 3/4 riser 2, 5/6 riser 3.
    VI_Local_Valve_Open : ARRAY[1..6] OF BOOL;
    VI_Local_Valve_Close : ARRAY[1..6] OF BOOL;
END_VAR
VAR
    L_i : INT;
END_VAR

FOR L_i := 1 TO GVL_CONSTANTS.C_MAX_WATER_ZONES DO
    GVL_WATER_OUTPUT.DO_Water_Zone_Enable[L_i] := VI_Zone_Enable[L_i];
END_FOR;

GVL_WATER_OUTPUT.DO_Water_Valve_35_Open := VI_Valve_35_Open;
GVL_WATER_OUTPUT.DO_Water_Valve_35_Close := VI_Valve_35_Close;
GVL_WATER_OUTPUT.DO_Water_Valve_36_Open := VI_Valve_36_Open;
GVL_WATER_OUTPUT.DO_Water_Valve_36_Close := VI_Valve_36_Close;

FOR L_i := 1 TO 6 DO
    GVL_WATER_OUTPUT.DO_Water_Local_Valve_Open[L_i] := VI_Local_Valve_Open[L_i];
    GVL_WATER_OUTPUT.DO_Water_Local_Valve_Close[L_i] := VI_Local_Valve_Close[L_i];
END_FOR;

END_FUNCTION_BLOCK
// >>> BULK_SYNC_ANCHOR: FB_Water_Output_Projection <<<

(* ---- FB_Water_Output_Projector.st ---- *)
FUNCTION_BLOCK FB_Water_Output_Projector
VAR_INPUT
    VI_Enable : BOOL;
    VI_System_Time_MS : UDINT;
END_VAR
VAR
    L_i : INT;
    L_Authority : ST_Water_Isolation_Authority_State;
    L_Valve : ST_Water_Valve_Runtime_State;
    L_Output : ST_Water_Output_Projection_State;
    L_Any_Projected : BOOL;
    L_Any_Denied : BOOL;
    L_Global_Fallback : BOOL;
END_VAR

IF NOT VI_Enable THEN
    GVL_Water_Output_Projection.G_Runtime_Valid := FALSE;
    RETURN;
END_IF;

L_Any_Projected := FALSE;
L_Any_Denied := FALSE;
L_Global_Fallback := FALSE;

FOR L_i := 1 TO GVL_CONSTANTS.C_MAX_FLOOD_SENSORS DO

    L_Authority := GVL_Water_Isolation_Authority.G_Authority_State[L_i];
    L_Valve := GVL_Water_Valve_Runtime.G_Valve_Runtime_State[L_i];

    // Reset all projection fields per sensor to prevent state leakage across loop iterations.
    L_Output.Projection_Valid := FALSE;
    L_Output.Projection_System_Time_MS := 0;
    L_Output.Output_Owner_Valid := FALSE;
    L_Output.Output_Owner_Id := 0;
    L_Output.Valve_Id := 0;
    L_Output.Valve_Group_Id := 0;
    L_Output.Selective_Authority_Allowed := FALSE;
    L_Output.Global_Fallback_Required := FALSE;
    L_Output.Authority_Valid := FALSE;
    L_Output.Physical_Close_Project := FALSE;
    L_Output.Physical_Open_Project := FALSE;
    L_Output.Expected_Closed := FALSE;
    L_Output.Expected_Open := FALSE;
    L_Output.Confirmed_Closed := FALSE;
    L_Output.Confirmed_Open := FALSE;
    L_Output.Confirmation_Unknown := FALSE;
    L_Output.Projection_Allowed := FALSE;
    L_Output.Projection_Denied := FALSE;
    L_Output.Projection_Code := 0;
    L_Output.Projection_Text := '';
    L_Output.Projection_Activated_Event := FALSE;
    L_Output.Projection_Denied_Event := FALSE;

    L_Output.Projection_Valid := TRUE;
    L_Output.Projection_System_Time_MS := VI_System_Time_MS;
    L_Output.Output_Owner_Valid := TRUE;
    L_Output.Output_Owner_Id := TO_UINT(L_i);
    L_Output.Valve_Id := L_Valve.Valve_Id;
    L_Output.Valve_Group_Id := L_Valve.Valve_Group_Id;
    L_Output.Selective_Authority_Allowed := L_Authority.Selective_Authority_Allowed;
    L_Output.Global_Fallback_Required := L_Authority.Global_Fallback_Required;
    L_Output.Authority_Valid := L_Authority.Decision_Valid;

    IF L_Output.Global_Fallback_Required THEN
        L_Output.Projection_Allowed := TRUE;
        L_Output.Physical_Close_Project := TRUE;
        L_Output.Expected_Closed := TRUE;
        L_Output.Projection_Code := 1;
        L_Output.Projection_Text := 'Global fallback output projection active';
        L_Global_Fallback := TRUE;
    ELSIF L_Output.Selective_Authority_Allowed AND L_Output.Authority_Valid THEN
        L_Output.Projection_Allowed := TRUE;
        L_Output.Physical_Close_Project := TRUE;
        L_Output.Expected_Closed := TRUE;
        L_Output.Projection_Code := 10;
        L_Output.Projection_Text := 'Selective authority output projection active';
    ELSE
        L_Output.Projection_Denied := TRUE;
        L_Output.Projection_Code := 100;
        L_Output.Projection_Text := 'Projection denied';
        L_Any_Denied := TRUE;
    END_IF;

    L_Output.Confirmed_Closed := L_Valve.Confirmed_Closed;
    L_Output.Confirmed_Open := L_Valve.Confirmed_Open;
    L_Output.Confirmation_Unknown := L_Valve.Confirmation_Unknown;
    L_Output.Projection_Activated_Event := L_Output.Projection_Allowed;
    L_Output.Projection_Denied_Event := L_Output.Projection_Denied;

    GVL_Water_Output_Projection.G_Output_Projection_State[L_i] := L_Output;
    L_Any_Projected := L_Any_Projected OR L_Output.Projection_Allowed;
END_FOR;

GVL_Water_Output_Projection.G_Any_Output_Projected := L_Any_Projected;
GVL_Water_Output_Projection.G_Any_Projection_Denied := L_Any_Denied;
GVL_Water_Output_Projection.G_Global_Fallback_Projecting := L_Global_Fallback;
GVL_Water_Output_Projection.G_Runtime_Valid := TRUE;
GVL_Water_Output_Projection.G_Last_Update_MS := VI_System_Time_MS;

IF L_Global_Fallback THEN
    GVL_Water_Output_Projection.G_Status_Code := 2;
    GVL_Water_Output_Projection.G_Status_Text := 'Global fallback output projection active';
ELSIF L_Any_Projected THEN
    GVL_Water_Output_Projection.G_Status_Code := 1;
    GVL_Water_Output_Projection.G_Status_Text := 'Selective output projection active';
ELSE
    GVL_Water_Output_Projection.G_Status_Code := 0;
    GVL_Water_Output_Projection.G_Status_Text := 'No output projections active';
END_IF;

END_FUNCTION_BLOCK
